  Call Extruder(12358.70300)
  MoveL 1243 to (-24.11, 11.61, 60) mm, rotated rx -180 ry 0 rz 180 deg; joints [-156.928, -57.132, -93.982, 25.942, 63.614, -12.2]
  Call Extruder(12368.06781)
  MoveL 1244 to (-26.09, 5.96, 60) mm, rotated rx -180 ry 0 rz 180 deg; joints [-157.665, -56.949, -94.65, 25.035, 63.9, -11.611]
  Call Extruder(12377.43291)
  MoveL 1245 to (-26.77, 0, 60) mm, rotated rx -180 ry 0 rz 180 deg; joints [-158.546, -56.823, -95.122, 24.004, 64.04, -11.03]
  Call Extruder(12382.22164)
  MoveL 1246 to (-26.42, -3.05, 60) mm, rotated rx -180 ry 0 rz 180 deg; joints [-159.044, -56.788, -95.251, 23.441, 64.033, -10.75]
  Set speed (130.0 mm/s)
  MoveL 1247 to (-41.86, -6.3, 60) mm, rotated rx 180 ry 0 rz 180 deg; joints [-158.606, -56.142, -97.794, 23.564, 65.852, -10.116]
  Call Extruder(12387.21949)
  Set speed (60.0 mm/s)
  MoveL 1248 to (-41.5, -9.47, 60) mm, rotated rx 180 ry 0 rz -180 deg; joints [-159.151, -56.11, -97.925, 22.957, 65.848, -9.832]
  Call Extruder(12402.11514)
  MoveL 1249 to (-38.36, -18.47, 60) mm, rotated rx -180 ry 0 rz 180 deg; joints [-160.835, -56.105, -97.945, 21.132, 65.585, -9.077]
  Call Extruder(12417.01100)
  MoveL 1250 to (-33.28, -26.54, 60) mm, rotated rx 180 ry 0 rz 180 deg; joints [-162.466, -56.194, -97.578, 19.403, 65.076, -8.443]
  Call Extruder(12431.90681)
  MoveL 1251 to (-26.54, -33.28, 60) mm, rotated rx -180 ry 0 rz -180 deg; joints [-163.93, -56.376, -96.846, 17.884, 64.347, -7.952]
  Call Extruder(12446.80266)
  MoveL 1252 to (-18.47, -38.36, 60) mm, rotated rx 180 ry 0 rz 180 deg; joints [-165.137, -56.645, -95.795, 16.666, 63.436, -7.625]
  Call Extruder(12461.69831)
  MoveL 1253 to (-9.47, -41.5, 60) mm, rotated rx 180 ry 0 rz 180 deg; joints [-166.024, -56.995, -94.483, 15.815, 62.396, -7.477]
  Call Extruder(12476.59419)
  MoveL 1254 to (0, -42.57, 60) mm, rotated rx 180 ry 0 rz 180 deg; joints [-166.562, -57.411, -92.984, 15.366, 61.283, -7.522]
  Call Extruder(12481.08976)
  MoveL 1255 to (2.86, -42.25, 60) mm, rotated rx 180 ry 0 rz 180 deg; joints [-166.618, -57.549, -92.502, 15.353, 60.943, -7.595]
  Call Extruder(12491.49006)
  MoveL 1256 to (9.47, -41.51, 60) mm, rotated rx 180 ry 0 rz 180 deg; joints [-166.745, -57.877, -91.377, 15.328, 60.158, -7.767]
  Call Extruder(12506.38572)
  MoveL 1257 to (18.47, -38.36, 60) mm, rotated rx -180 ry 0 rz 180 deg; joints [-166.591, -58.369, -89.743, 15.683, 59.079, -8.21]
  Call Extruder(12521.28157)
  MoveL 1258 to (26.54, -33.28, 60) mm, rotated rx 180 ry 0 rz 180 deg; joints [-166.133, -58.862, -88.162, 16.398, 58.102, -8.839]
  Call Extruder(12536.17739)
  MoveL 1259 to (33.29, -26.54, 60) mm, rotated rx -180 ry 0 rz 180 deg; joints [-165.409, -59.329, -86.71, 17.424, 57.275, -9.629]
  Call Extruder(12551.07324)
  MoveL 1260 to (38.36, -18.47, 60) mm, rotated rx -180 ry 0 rz -180 deg; joints [-164.468, -59.742, -85.455, 18.7, 56.639, -10.544]
  Call Extruder(12565.96889)
  MoveL 1261 to (41.5, -9.47, 60) mm, rotated rx 180 ry 0 rz 180 deg; joints [-163.355, -60.078, -84.454, 20.158, 56.225, -11.534]
  Call Extruder(12580.86476)
  MoveL 1262 to (42.57, 0, 60) mm, rotated rx 180 ry 0 rz 180 deg; joints [-162.12, -60.316, -83.753, 21.723, 56.051, -12.544]
  Call Extruder(12595.76064)
  MoveL 1263 to (41.51, 9.47, 60) mm, rotated rx 180 ry 0 rz 180 deg; joints [-160.81, -60.442, -83.386, 23.323, 56.123, -13.513]
  Call Extruder(12610.65630)
  MoveL 1264 to (38.36, 18.47, 60) mm, rotated rx -180 ry 0 rz -180 deg; joints [-159.475, -60.448, -83.368, 24.884, 56.434, -14.384]
  Call Extruder(12625.55214)
  MoveL 1265 to (33.29, 26.54, 60) mm, rotated rx 180 ry 0 rz 180 deg; joints [-158.16, -60.334, -83.702, 26.343, 56.966, -15.106]
  Call Extruder(12640.44797)
  MoveL 1266 to (26.54, 33.28, 60) mm, rotated rx 180 ry 0 rz -180 deg; joints [-156.916, -60.106, -84.37, 27.64, 57.689, -15.638]
  Call Extruder(12655.34381)
  MoveL 1267 to (18.47, 38.36, 60) mm, rotated rx 180 ry 0 rz -180 deg; joints [-155.789, -59.779, -85.343, 28.727, 58.565, -15.953]
  Call Extruder(12670.23948)
  MoveL 1268 to (9.47, 41.51, 60) mm, rotated rx 180 ry 0 rz 180 deg; joints [-154.828, -59.372, -86.576, 29.563, 59.552, -16.037]
  Call Extruder(12685.13535)
  MoveL 1269 to (0, 42.57, 60) mm, rotated rx 180 ry 0 rz 180 deg; joints [-154.081, -58.91, -88.012, 30.113, 60.601, -15.892]
  Call Extruder(12700.03122)
  MoveL 1270 to (-9.47, 41.51, 60) mm, rotated rx 180 ry 0 rz -180 deg; joints [-153.594, -58.418, -89.583, 30.349, 61.666, -15.53]
  Call Extruder(12714.92687)
  MoveL 1271 to (-18.47, 38.36, 60) mm, rotated rx 180 ry 0 rz 180 deg; joints [-153.408, -57.925, -91.215, 30.248, 62.698, -14.975]
  Call Extruder(12729.82273)
  MoveL 1272 to (-26.54, 33.29, 60) mm, rotated rx 180 ry 0 rz 180 deg; joints [-153.557, -57.456, -92.828, 29.797, 63.651, -14.261]
  Call Extruder(12744.71854)
  MoveL 1273 to (-33.28, 26.54, 60) mm, rotated rx 180 ry 0 rz -180 deg; joints [-154.059, -57.033, -94.341, 28.995, 64.481, -13.428]
  Call Extruder(12759.61439)
  MoveL 1274 to (-38.36, 18.47, 60) mm, rotated rx 180 ry 0 rz -180 deg; joints [-154.913, -56.677, -95.675, 27.857, 65.148, -12.523]
  Call Extruder(12774.51005)
  MoveL 1275 to (-41.51, 9.47, 60) mm, rotated rx 180 ry 0 rz -180 deg; joints [-156.091, -56.399, -96.755, 26.422, 65.617, -11.593]
  Call Extruder(12789.40592)
  MoveL 1276 to (-42.57, 0, 60) mm, rotated rx 180 ry 0 rz -180 deg; joints [-157.533, -56.208, -97.521, 24.758, 65.857, -10.682]
  Call Extruder(12796.96020)
  MoveL 1277 to (-42.03, -4.8, 60) mm, rotated rx 180 ry 0 rz 180 deg; joints [-158.35, -56.157, -97.731, 23.848, 65.853, -10.25]
  Set speed (130.0 mm/s)
  MoveL 1278 to (-54.1, -7.67, 60) mm, rotated rx 180 ry 0 rz 180 deg; joints [-158.024, -55.698, -99.697, 23.934, 67.287, -9.724]
  Call Extruder(12801.03283)
  Set speed (30.0 mm/s)
  MoveL 1279 to (-53.59, -12.23, 60) mm, rotated rx -180 ry 0 rz 180 deg; joints [-158.835, -55.656, -99.887, 23.042, 67.288, -9.326]
  Call Extruder(12811.96296)
  MoveL 1280 to (-49.53, -23.85, 60) mm, rotated rx 180 ry 0 rz -180 deg; joints [-161.095, -55.65, -99.912, 20.615, 66.959, -8.375]
  Call Extruder(12822.89325)
  MoveL 1281 to (-42.98, -34.27, 60) mm, rotated rx -180 ry 0 rz 180 deg; joints [-163.275, -55.758, -99.429, 18.317, 66.303, -7.579]
  Call Extruder(12833.82337)
  MoveL 1282 to (-34.27, -42.98, 60) mm, rotated rx 180 ry 0 rz -180 deg; joints [-165.21, -55.98, -98.468, 16.312, 65.352, -6.958]
  Call Extruder(12844.75365)
  MoveL 1283 to (-23.85, -49.53, 60) mm, rotated rx 180 ry 0 rz 180 deg; joints [-166.774, -56.315, -97.09, 14.727, 64.164, -6.535]
  Call Extruder(12855.68378)
  MoveL 1284 to (-12.23, -53.59, 60) mm, rotated rx 180 ry 0 rz 180 deg; joints [-167.889, -56.754, -95.38, 13.644, 62.807, -6.33]
  Call Extruder(12866.61401)
  MoveL 1285 to (0, -54.97, 60) mm, rotated rx 180 ry 0 rz 180 deg; joints [-168.526, -57.284, -93.434, 13.1, 61.358, -6.365]
  Call Extruder(12870.40133)
  MoveL 1286 to (4.24, -54.49, 60) mm, rotated rx -180 ry 0 rz 180 deg; joints [-168.587, -57.487, -92.718, 13.096, 60.852, -6.464]
  Call Extruder(12877.54423)
  MoveL 1287 to (12.23, -53.59, 60) mm, rotated rx 180 ry 0 rz 180 deg; joints [-168.697, -57.883, -91.355, 13.094, 59.898, -6.654]
  Call Extruder(12888.47437)
  MoveL 1288 to (23.85, -49.53, 60) mm, rotated rx 180 ry 0 rz 180 deg; joints [-168.436, -58.521, -89.25, 13.597, 58.501, -7.203]
  Call Extruder(12899.40465)
  MoveL 1289 to (34.27, -42.98, 60) mm, rotated rx 180 ry 0 rz 180 deg; joints [-167.797, -59.164, -87.217, 14.558, 57.238, -8]
  Call Extruder(12910.33477)
  MoveL 1290 to (42.98, -34.27, 60) mm, rotated rx -180 ry 0 rz 180 deg; joints [-166.837, -59.776, -85.354, 15.91, 56.172, -9.017]
  Call Extruder(12921.26505)
  MoveL 1291 to (49.53, -23.85, 60) mm, rotated rx 180 ry 0 rz 180 deg; joints [-165.618, -60.319, -83.744, 17.573, 55.354, -10.206]
  Call Extruder(12932.19519)
  MoveL 1292 to (53.59, -12.23, 60) mm, rotated rx 180 ry 0 rz -180 deg; joints [-164.2, -60.762, -82.461, 19.457, 54.825, -11.504]
  Call Extruder(12943.12541)
  MoveL 1293 to (54.97, 0, 60) mm, rotated rx -180 ry 0 rz 180 deg; joints [-162.641, -61.077, -81.564, 21.469, 54.608, -12.832]
  Call Extruder(12954.05563)
  MoveL 1294 to (53.59, 12.23, 60) mm, rotated rx 180 ry 0 rz -180 deg; joints [-160.996, -61.244, -81.093, 23.512, 54.71, -14.109]
  Call Extruder(12964.98577)
  MoveL 1295 to (49.52, 23.85, 60) mm, rotated rx 180 ry 0 rz -180 deg; joints [-159.322, -61.252, -81.071, 25.495, 55.121, -15.253]
  Call Extruder(12975.91605)
  MoveL 1296 to (42.98, 34.27, 60) mm, rotated rx -180 ry 0 rz 180 deg; joints [-157.673, -61.1, -81.498, 27.338, 55.815, -16.197]
  Call Extruder(12986.84617)
  MoveL 1297 to (34.27, 42.98, 60) mm, rotated rx 180 ry 0 rz 180 deg; joints [-156.102, -60.8, -82.354, 28.973, 56.752, -16.887]
  Call Extruder(12997.77645)
  MoveL 1298 to (23.85, 49.52, 60) mm, rotated rx 180 ry 0 rz 180 deg; joints [-154.667, -60.368, -83.601, 30.344, 57.883, -17.287]
  Call Extruder(13008.70659)
  MoveL 1299 to (12.23, 53.59, 60) mm, rotated rx -180 ry 0 rz 180 deg; joints [-153.426, -59.833, -85.181, 31.405, 59.15, -17.384]
  Call Extruder(13019.63681)
  MoveL 1300 to (0, 54.97, 60) mm, rotated rx 180 ry 0 rz 180 deg; joints [-152.438, -59.227, -87.023, 32.118, 60.494, -17.18]
  Call Extruder(13030.56704)
  MoveL 1301 to (-12.23, 53.59, 60) mm, rotated rx 180 ry 0 rz 180 deg; joints [-151.764, -58.585, -89.043, 32.449, 61.856, -16.695]
  Call Extruder(13041.49717)
  MoveL 1302 to (-23.85, 49.52, 60) mm, rotated rx 180 ry 0 rz 180 deg; joints [-151.463, -57.945, -91.146, 32.366, 63.175, -15.961]
  Call Extruder(13052.42745)
  MoveL 1303 to (-34.27, 42.98, 60) mm, rotated rx -180 ry 0 rz 180 deg; joints [-151.589, -57.341, -93.232, 31.843, 64.397, -15.023]
  Call Extruder(13063.35757)
  MoveL 1304 to (-42.98, 34.27, 60) mm, rotated rx 180 ry 0 rz -180 deg; joints [-152.179, -56.803, -95.196, 30.865, 65.467, -13.937]
  Call Extruder(13074.28785)
  MoveL 1305 to (-49.52, 23.85, 60) mm, rotated rx 180 ry 0 rz 180 deg; joints [-153.248, -56.354, -96.934, 29.437, 66.335, -12.763]
  Call Extruder(13085.21799)
  MoveL 1306 to (-53.59, 12.23, 60) mm, rotated rx -180 ry 0 rz 180 deg; joints [-154.769, -56.009, -98.348, 27.596, 66.954, -11.565]
  Call Extruder(13096.14821)
  MoveL 1307 to (-54.97, 0, 60) mm, rotated rx 180 ry 0 rz -180 deg; joints [-156.673, -55.775, -99.354, 25.423, 67.282, -10.402]
  Call Extruder(13101.67383)
  MoveL 1308 to (-54.27, -6.18, 60) mm, rotated rx 180 ry 0 rz -180 deg; joints [-157.76, -55.712, -99.633, 24.224, 67.287, -9.855]
  Set speed (130.0 mm/s)
  MoveL 1309 to (-49.9, -9.51, 60) mm, rotated rx 180 ry 0 rz 180 deg; joints [-158.616, -55.814, -99.183, 23.367, 66.823, -9.65]
  MoveL 1310 to (2.97, -12.99, 60) mm, rotated rx 180 ry 0 rz -180 deg; joints [-162.152, -57.947, -91.141, 20.571, 60.725, -10.399]
  Call Extruder(13106.33740)
  Set speed (80.0 mm/s)
  MoveL 1311 to (5.78, -12.01, 60) mm, rotated rx 180 ry 0 rz -180 deg; joints [-162.141, -58.1, -90.629, 20.655, 60.391, -10.551]
  Call Extruder(13111.00102)
  MoveL 1312 to (8.31, -10.42, 60) mm, rotated rx 180 ry 0 rz -180 deg; joints [-162.027, -58.251, -90.129, 20.855, 60.086, -10.757]
  Call Extruder(13115.66521)
  MoveL 1313 to (10.42, -8.31, 60) mm, rotated rx -180 ry 0 rz 180 deg; joints [-161.819, -58.392, -89.668, 21.157, 59.827, -11.007]
  Call Extruder(13120.32884)
  MoveL 1314 to (12.01, -5.78, 60) mm, rotated rx 180 ry 0 rz 180 deg; joints [-161.529, -58.516, -89.267, 21.546, 59.625, -11.291]
  Call Extruder(13124.99241)
  MoveL 1315 to (12.99, -2.97, 60) mm, rotated rx 180 ry 0 rz -180 deg; joints [-161.171, -58.615, -88.947, 22, 59.491, -11.592]
  Call Extruder(13129.65636)
  MoveL 1316 to (13.33, 0, 60) mm, rotated rx -180 ry 0 rz 180 deg; joints [-160.763, -58.686, -88.723, 22.499, 59.431, -11.895]
  Call Extruder(13134.32032)
  MoveL 1317 to (12.99, 2.97, 60) mm, rotated rx 180 ry 0 rz 180 deg; joints [-160.324, -58.723, -88.605, 23.016, 59.448, -12.185]
  Call Extruder(13138.98389)
  MoveL 1318 to (12.01, 5.78, 60) mm, rotated rx -180 ry 0 rz -180 deg; joints [-159.874, -58.724, -88.599, 23.527, 59.541, -12.446]
  Call Extruder(13143.64751)
  MoveL 1319 to (10.42, 8.31, 60) mm, rotated rx -180 ry 0 rz 180 deg; joints [-159.432, -58.691, -88.706, 24.009, 59.704, -12.664]
  Call Extruder(13148.31170)
  MoveL 1320 to (8.31, 10.42, 60) mm, rotated rx -180 ry 0 rz 180 deg; joints [-159.021, -58.624, -88.92, 24.438, 59.929, -12.828]
  Call Extruder(13152.97533)
  MoveL 1321 to (5.78, 12.01, 60) mm, rotated rx 180 ry 0 rz 180 deg; joints [-158.657, -58.527, -89.232, 24.796, 60.205, -12.929]
  Call Extruder(13157.63890)
  MoveL 1322 to (2.97, 12.99, 60) mm, rotated rx -180 ry 0 rz 180 deg; joints [-158.359, -58.405, -89.625, 25.065, 60.518, -12.962]
  Call Extruder(13162.30285)
  MoveL 1323 to (0, 13.33, 60) mm, rotated rx -180 ry 0 rz 180 deg; joints [-158.143, -58.266, -90.082, 25.231, 60.853, -12.926]
  Call Extruder(13166.96681)
  MoveL 1324 to (-2.97, 12.99, 60) mm, rotated rx 180 ry 0 rz 180 deg; joints [-158.019, -58.115, -90.578, 25.287, 61.194, -12.824]
  Call Extruder(13171.63038)
  MoveL 1325 to (-5.78, 12.01, 60) mm, rotated rx 180 ry 0 rz -180 deg; joints [-157.997, -57.962, -91.091, 25.228, 61.524, -12.661]
  Call Extruder(13176.29401)
  MoveL 1326 to (-8.31, 10.42, 60) mm, rotated rx 180 ry 0 rz 180 deg; joints [-158.08, -57.813, -91.593, 25.055, 61.826, -12.447]
  Call Extruder(13180.95820)
  MoveL 1327 to (-10.42, 8.31, 60) mm, rotated rx 180 ry 0 rz 180 deg; joints [-158.266, -57.677, -92.061, 24.774, 62.086, -12.192]
  Call Extruder(13185.62182)
  MoveL 1328 to (-12.01, 5.78, 60) mm, rotated rx 180 ry 0 rz -180 deg; joints [-158.549, -57.558, -92.469, 24.399, 62.291, -11.91]
  Call Extruder(13190.28539)
  MoveL 1329 to (-12.99, 2.97, 60) mm, rotated rx 180 ry 0 rz -180 deg; joints [-158.913, -57.464, -92.797, 23.946, 62.431, -11.615]
  Call Extruder(13194.94935)
  MoveL 1330 to (-13.33, 0, 60) mm, rotated rx 180 ry 0 rz -180 deg; joints [-159.341, -57.399, -93.028, 23.438, 62.497, -11.321]
  Call Extruder(13199.61330)
  MoveL 1331 to (-12.99, -2.97, 60) mm, rotated rx 180 ry 0 rz 180 deg; joints [-159.811, -57.364, -93.15, 22.901, 62.486, -11.042]
  Call Extruder(13204.27687)
  MoveL 1332 to (-12.01, -5.78, 60) mm, rotated rx 180 ry 0 rz -180 deg; joints [-160.294, -57.363, -93.156, 22.364, 62.398, -10.793]
  Call Extruder(13208.94050)
  MoveL 1333 to (-10.42, -8.31, 60) mm, rotated rx 180 ry 0 rz -180 deg; joints [-160.766, -57.394, -93.045, 21.856, 62.238, -10.583]
  Call Extruder(13213.60468)
  MoveL 1334 to (-8.31, -10.42, 60) mm, rotated rx 180 ry 0 rz -180 deg; joints [-161.2, -57.457, -92.825, 21.405, 62.012, -10.423]
  Call Extruder(13218.26832)
  MoveL 1335 to (-5.78, -12.01, 60) mm, rotated rx 180 ry 0 rz 180 deg; joints [-161.572, -57.548, -92.506, 21.034, 61.732, -10.322]
  Call Extruder(13222.93188)
  MoveL 1336 to (-2.97, -13, 60) mm, rotated rx 180 ry 0 rz 180 deg; joints [-161.863, -57.664, -92.104, 20.764, 61.414, -10.282]
  Call Extruder(13227.59582)
  MoveL 1337 to (0, -13.33, 60) mm, rotated rx -180 ry 0 rz -180 deg; joints [-162.059, -57.799, -91.642, 20.607, 61.072, -10.308]
  Call Extruder(13232.25979)
  MoveL 1338 to (2.97, -12.99, 60) mm, rotated rx 180 ry 0 rz -180 deg; joints [-162.152, -57.947, -91.141, 20.571, 60.725, -10.399]
  Set speed (130.0 mm/s)
  MoveL 1339 to (2.97, -12.99, 65) mm, rotated rx -180 ry 0 rz -180 deg; joints [-162.152, -57.18, -91.526, 20.647, 60.368, -10.553]
  MoveL 1340 to (-26.25, -4.54, 65) mm, rotated rx -180 ry 0 rz 180 deg; joints [-159.288, -55.977, -95.706, 23.243, 63.66, -10.789]
  Call Extruder(13234.49242)
  Set speed (60.0 mm/s)
  MoveL 1341 to (-26.09, -5.96, 65) mm, rotated rx 180 ry 0 rz 180 deg; joints [-159.522, -55.961, -95.763, 22.979, 63.655, -10.657]
  Call Extruder(13243.85722)
  MoveL 1342 to (-24.12, -11.61, 65) mm, rotated rx 180 ry 0 rz 180 deg; joints [-160.532, -55.958, -95.775, 21.869, 63.481, -10.16]
  Call Extruder(13253.22213)
  MoveL 1343 to (-20.93, -16.69, 65) mm, rotated rx 180 ry 0 rz -180 deg; joints [-161.513, -56.02, -95.549, 20.817, 63.158, -9.741]
  Call Extruder(13262.58734)
  MoveL 1344 to (-16.69, -20.93, 65) mm, rotated rx 180 ry 0 rz 180 deg; joints [-162.406, -56.144, -95.098, 19.886, 62.702, -9.419]
  Call Extruder(13271.95226)
  MoveL 1345 to (-11.61, -24.12, 65) mm, rotated rx 180 ry 0 rz 180 deg; joints [-163.159, -56.325, -94.447, 19.129, 62.138, -9.207]
  Call Extruder(13281.31705)
  MoveL 1346 to (-5.96, -26.09, 65) mm, rotated rx 180 ry 0 rz -180 deg; joints [-163.733, -56.558, -93.631, 18.587, 61.495, -9.118]
  Call Extruder(13290.68216)
  MoveL 1347 to (0, -26.77, 65) mm, rotated rx 180 ry 0 rz -180 deg; joints [-164.103, -56.831, -92.694, 18.286, 60.806, -9.156]
  Call Extruder(13293.06822)
  MoveL 1348 to (1.52, -26.59, 65) mm, rotated rx 180 ry 0 rz -180 deg; joints [-164.143, -56.907, -92.438, 18.273, 60.629, -9.199]
  Call Extruder(13300.04726)
  MoveL 1349 to (5.96, -26.09, 65) mm, rotated rx 180 ry 0 rz 180 deg; joints [-164.258, -57.133, -91.685, 18.236, 60.109, -9.325]
  Call Extruder(13309.41206)
  MoveL 1350 to (11.61, -24.11, 65) mm, rotated rx 180 ry 0 rz 180 deg; joints [-164.201, -57.447, -90.654, 18.433, 59.439, -9.618]
  Call Extruder(13318.77697)
  MoveL 1351 to (16.69, -20.93, 65) mm, rotated rx -180 ry 0 rz 180 deg; joints [-163.944, -57.76, -89.654, 18.859, 58.831, -10.026]
  Call Extruder(13328.14218)
  MoveL 1352 to (20.93, -16.69, 65) mm, rotated rx 180 ry 0 rz 180 deg; joints [-163.508, -58.053, -88.733, 19.488, 58.316, -10.529]
  Call Extruder(13337.50710)
  MoveL 1353 to (24.12, -11.61, 65) mm, rotated rx 180 ry 0 rz 180 deg; joints [-162.92, -58.311, -87.934, 20.283, 57.918, -11.105]
  Call Extruder(13346.87189)
  MoveL 1354 to (26.09, -5.96, 65) mm, rotated rx -180 ry 0 rz -180 deg; joints [-162.209, -58.52, -87.297, 21.201, 57.659, -11.723]
  Call Extruder(13356.23700)
  MoveL 1355 to (26.77, 0, 65) mm, rotated rx -180 ry 0 rz -180 deg; joints [-161.41, -58.668, -86.851, 22.197, 57.548, -12.35]
  Call Extruder(13365.60210)
  MoveL 1356 to (26.09, 5.96, 65) mm, rotated rx 180 ry 0 rz 180 deg; joints [-160.556, -58.746, -86.617, 23.222, 57.591, -12.951]
  Call Extruder(13374.96690)
  MoveL 1357 to (24.12, 11.61, 65) mm, rotated rx 180 ry 0 rz 180 deg; joints [-159.683, -58.75, -86.606, 24.23, 57.784, -13.492]
  Call Extruder(13384.33181)
  MoveL 1358 to (20.93, 16.69, 65) mm, rotated rx 180 ry 0 rz 180 deg; joints [-158.826, -58.679, -86.818, 25.176, 58.116, -13.943]
  Call Extruder(13393.69702)
  MoveL 1359 to (16.69, 20.93, 65) mm, rotated rx -180 ry 0 rz 180 deg; joints [-158.019, -58.538, -87.244, 26.018, 58.569, -14.281]
  Call Extruder(13403.06194)
  MoveL 1360 to (11.61, 24.11, 65) mm, rotated rx 180 ry 0 rz -180 deg; joints [-157.299, -58.335, -87.863, 26.722, 59.121, -14.487]
  Call Extruder(13412.42674)
  MoveL 1361 to (5.96, 26.09, 65) mm, rotated rx -180 ry 0 rz 180 deg; joints [-156.697, -58.081, -88.647, 27.257, 59.744, -14.552]
  Call Extruder(13421.79184)
  MoveL 1362 to (0, 26.77, 65) mm, rotated rx -180 ry 0 rz 180 deg; joints [-156.245, -57.79, -89.558, 27.597, 60.408, -14.474]
  Call Extruder(13431.15695)
  MoveL 1363 to (-5.96, 26.09, 65) mm, rotated rx 180 ry 0 rz 180 deg; joints [-155.969, -57.479, -90.553, 27.726, 61.082, -14.26]
  Call Extruder(13440.52174)
  MoveL 1364 to (-11.61, 24.12, 65) mm, rotated rx 180 ry 0 rz 180 deg; joints [-155.891, -57.163, -91.582, 27.631, 61.733, -13.923]
  Call Extruder(13449.88666)
  MoveL 1365 to (-16.69, 20.93, 65) mm, rotated rx 180 ry 0 rz -180 deg; joints [-156.025, -56.86, -92.596, 27.31, 62.332, -13.483]
  Call Extruder(13459.25187)
  MoveL 1366 to (-20.93, 16.69, 65) mm, rotated rx 180 ry 0 rz -180 deg; joints [-156.374, -56.583, -93.543, 26.77, 62.849, -12.964]
  Call Extruder(13468.61678)
  MoveL 1367 to (-24.11, 11.61, 65) mm, rotated rx -180 ry 0 rz 180 deg; joints [-156.928, -56.346, -94.373, 26.029, 63.258, -12.394]
  Call Extruder(13477.98158)
  MoveL 1368 to (-26.09, 5.96, 65) mm, rotated rx -180 ry 0 rz -180 deg; joints [-157.665, -56.159, -95.042, 25.119, 63.538, -11.8]
  Call Extruder(13487.34669)
  MoveL 1369 to (-26.77, 0, 65) mm, rotated rx -180 ry 0 rz 180 deg; joints [-158.546, -56.029, -95.514, 24.084, 63.674, -11.212]
  Call Extruder(13492.13541)
  MoveL 1370 to (-26.42, -3.05, 65) mm, rotated rx 180 ry 0 rz -180 deg; joints [-159.044, -55.994, -95.644, 23.52, 63.665, -10.928]
  Set speed (130.0 mm/s)
  MoveL 1371 to (-41.86, -6.29, 65) mm, rotated rx 180 ry 0 rz 180 deg; joints [-158.606, -55.328, -98.193, 23.639, 65.471, -10.299]
  Call Extruder(13497.13327)
  Set speed (60.0 mm/s)
  MoveL 1372 to (-41.51, -9.47, 65) mm, rotated rx -180 ry 0 rz 180 deg; joints [-159.151, -55.295, -98.325, 23.031, 65.466, -10.011]
  Call Extruder(13512.02892)
  MoveL 1373 to (-38.36, -18.47, 65) mm, rotated rx 180 ry 0 rz -180 deg; joints [-160.835, -55.29, -98.344, 21.201, 65.198, -9.242]
  Call Extruder(13526.92477)
  MoveL 1374 to (-33.28, -26.54, 65) mm, rotated rx 180 ry 0 rz 180 deg; joints [-162.466, -55.382, -97.976, 19.468, 64.686, -8.595]
  Call Extruder(13541.82058)
  MoveL 1375 to (-26.54, -33.28, 65) mm, rotated rx 180 ry 0 rz -180 deg; joints [-163.93, -55.569, -97.243, 17.945, 63.956, -8.093]
  Call Extruder(13556.71644)
  MoveL 1376 to (-18.47, -38.36, 65) mm, rotated rx 180 ry 0 rz 180 deg; joints [-165.137, -55.847, -96.189, 16.724, 63.048, -7.755]
  Call Extruder(13571.61209)
  MoveL 1377 to (-9.47, -41.51, 65) mm, rotated rx 180 ry 0 rz -180 deg; joints [-166.024, -56.206, -94.874, 15.872, 62.013, -7.6]
  Call Extruder(13586.50797)
  MoveL 1378 to (0, -42.57, 65) mm, rotated rx 180 ry 0 rz 180 deg; joints [-166.562, -56.633, -93.372, 15.423, 60.906, -7.64]
  Call Extruder(13591.65957)
  MoveL 1379 to (3.28, -42.2, 65) mm, rotated rx 180 ry 0 rz 180 deg; joints [-166.626, -56.795, -92.818, 15.409, 60.52, -7.724]
  Call Extruder(13601.40384)
  MoveL 1380 to (9.47, -41.51, 65) mm, rotated rx 180 ry 0 rz 180 deg; joints [-166.745, -57.109, -91.762, 15.386, 59.789, -7.884]
  Call Extruder(13616.29950)
  MoveL 1381 to (18.47, -38.36, 65) mm, rotated rx -180 ry 0 rz 180 deg; joints [-166.591, -57.612, -90.126, 15.744, 58.718, -8.328]
  Call Extruder(13631.19534)
  MoveL 1382 to (26.54, -33.28, 65) mm, rotated rx 180 ry 0 rz 180 deg; joints [-166.133, -58.114, -88.543, 16.463, 57.749, -8.961]
  Call Extruder(13646.09116)
  MoveL 1383 to (33.28, -26.54, 65) mm, rotated rx 180 ry 0 rz 180 deg; joints [-165.409, -58.589, -87.089, 17.494, 56.93, -9.758]
  Call Extruder(13660.98702)
  MoveL 1384 to (38.36, -18.47, 65) mm, rotated rx 180 ry 0 rz 180 deg; joints [-164.468, -59.009, -85.832, 18.776, 56.302, -10.681]
  Call Extruder(13675.88267)
  MoveL 1385 to (41.5, -9.47, 65) mm, rotated rx -180 ry 0 rz 180 deg; joints [-163.355, -59.35, -84.83, 20.239, 55.895, -11.681]
  Call Extruder(13690.77854)
  MoveL 1386 to (42.57, 0, 65) mm, rotated rx 180 ry 0 rz -180 deg; joints [-162.12, -59.592, -84.129, 21.811, 55.727, -12.7]
  Call Extruder(13705.67441)
  MoveL 1387 to (41.5, 9.47, 65) mm, rotated rx -180 ry 0 rz 180 deg; joints [-160.81, -59.72, -83.762, 23.415, 55.805, -13.679]
  Call Extruder(13720.57008)
  MoveL 1388 to (38.36, 18.47, 65) mm, rotated rx -180 ry 0 rz 180 deg; joints [-159.475, -59.726, -83.744, 24.982, 56.12, -14.56]
  Call Extruder(13735.46592)
  MoveL 1389 to (33.28, 26.54, 65) mm, rotated rx -180 ry 0 rz 180 deg; joints [-158.16, -59.61, -84.078, 26.444, 56.655, -15.29]
  Call Extruder(13750.36174)
  MoveL 1390 to (26.54, 33.28, 65) mm, rotated rx -180 ry 0 rz 180 deg; joints [-156.916, -59.379, -84.747, 27.744, 57.379, -15.831]
  Call Extruder(13765.25759)
  MoveL 1391 to (18.47, 38.36, 65) mm, rotated rx 180 ry 0 rz -180 deg; joints [-155.789, -59.047, -85.721, 28.832, 58.254, -16.153]
  Call Extruder(13780.15325)
  MoveL 1392 to (9.47, 41.51, 65) mm, rotated rx 180 ry 0 rz -180 deg; joints [-154.828, -58.634, -86.955, 29.668, 59.238, -16.244]
  Call Extruder(13795.04912)
  MoveL 1393 to (0, 42.57, 65) mm, rotated rx 180 ry 0 rz -180 deg; joints [-154.081, -58.163, -88.392, 30.218, 60.284, -16.104]
  Call Extruder(13809.94500)
  MoveL 1394 to (-9.47, 41.51, 65) mm, rotated rx -180 ry 0 rz -180 deg; joints [-153.594, -57.662, -89.965, 30.451, 61.343, -15.745]
  Call Extruder(13824.84065)
  MoveL 1395 to (-18.47, 38.36, 65) mm, rotated rx 180 ry 0 rz 180 deg; joints [-153.408, -57.158, -91.6, 30.348, 62.368, -15.192]
  Call Extruder(13839.73650)
  MoveL 1396 to (-26.54, 33.29, 65) mm, rotated rx -180 ry 0 rz 180 deg; joints [-153.557, -56.678, -93.216, 29.894, 63.313, -14.477]
  Call Extruder(13854.63232)
  MoveL 1397 to (-33.28, 26.54, 65) mm, rotated rx -180 ry 0 rz 180 deg; joints [-154.059, -56.245, -94.732, 29.088, 64.134, -13.642]
  Call Extruder(13869.52817)
  MoveL 1398 to (-38.36, 18.47, 65) mm, rotated rx 180 ry 0 rz -180 deg; joints [-154.913, -55.879, -96.069, 27.945, 64.791, -12.732]
  Call Extruder(13884.42383)
  MoveL 1399 to (-41.5, 9.47, 65) mm, rotated rx 180 ry 0 rz 180 deg; joints [-156.091, -55.593, -97.152, 26.506, 65.25, -11.793]
  Call Extruder(13899.31970)
  MoveL 1400 to (-42.57, 0, 65) mm, rotated rx -180 ry 0 rz -180 deg; joints [-157.533, -55.396, -97.919, 24.836, 65.481, -10.873]
  Call Extruder(13906.87397)
  MoveL 1401 to (-42.03, -4.8, 65) mm, rotated rx -180 ry 0 rz 180 deg; joints [-158.35, -55.343, -98.13, 23.924, 65.474, -10.434]
  Set speed (130.0 mm/s)
  MoveL 1402 to (-54.1, -7.67, 65) mm, rotated rx -180 ry 0 rz 180 deg; joints [-158.024, -54.868, -100.101, 24.007, 66.899, -9.912]
  Call Extruder(13910.94661)
  Set speed (30.0 mm/s)
  MoveL 1403 to (-53.59, -12.23, 65) mm, rotated rx -180 ry 0 rz 180 deg; joints [-158.835, -54.824, -100.292, 23.112, 66.896, -9.507]
  Call Extruder(13921.87674)
  MoveL 1404 to (-49.52, -23.85, 65) mm, rotated rx 180 ry 0 rz 180 deg; joints [-161.095, -54.819, -100.317, 20.68, 66.56, -8.539]
  Call Extruder(13932.80702)
  MoveL 1405 to (-42.98, -34.27, 65) mm, rotated rx 180 ry 0 rz 180 deg; joints [-163.275, -54.931, -99.832, 18.376, 65.9, -7.725]
  Call Extruder(13943.73714)
  MoveL 1406 to (-34.27, -42.98, 65) mm, rotated rx 180 ry 0 rz -180 deg; joints [-165.21, -55.161, -98.868, 16.366, 64.95, -7.088]
  Call Extruder(13954.66743)
  MoveL 1407 to (-23.85, -49.53, 65) mm, rotated rx 180 ry 0 rz 180 deg; joints [-166.774, -55.506, -97.488, 14.778, 63.766, -6.651]
  Call Extruder(13965.59756)
  MoveL 1408 to (-12.23, -53.59, 65) mm, rotated rx -180 ry 0 rz 180 deg; joints [-167.889, -55.959, -95.773, 13.693, 62.415, -6.437]
  Call Extruder(13976.52778)
  MoveL 1409 to (0, -54.97, 65) mm, rotated rx -180 ry 0 rz 180 deg; joints [-168.526, -56.503, -93.823, 13.149, 60.976, -6.466]
  Call Extruder(13980.68794)
  MoveL 1410 to (4.65, -54.44, 65) mm, rotated rx -180 ry 0 rz 180 deg; joints [-168.593, -56.731, -93.035, 13.145, 60.424, -6.575]
  Call Extruder(13987.45800)
  MoveL 1411 to (12.23, -53.59, 65) mm, rotated rx 180 ry 0 rz 180 deg; joints [-168.697, -57.116, -91.741, 13.145, 59.525, -6.755]
  Call Extruder(13998.38814)
  MoveL 1412 to (23.85, -49.53, 65) mm, rotated rx -180 ry 0 rz 180 deg; joints [-168.436, -57.767, -89.632, 13.651, 58.139, -7.306]
  Call Extruder(14009.31842)
  MoveL 1413 to (34.27, -42.98, 65) mm, rotated rx -180 ry 0 rz 180 deg; joints [-167.797, -58.422, -87.597, 14.617, 56.887, -8.109]
  Call Extruder(14020.24854)
  MoveL 1414 to (42.98, -34.27, 65) mm, rotated rx -180 ry 0 rz 180 deg; joints [-166.837, -59.043, -85.731, 15.975, 55.831, -9.134]
  Call Extruder(14031.17883)
  MoveL 1415 to (49.52, -23.85, 65) mm, rotated rx -180 ry 0 rz 180 deg; joints [-165.618, -59.596, -84.12, 17.646, 55.023, -10.334]
  Call Extruder(14042.10896)
  MoveL 1416 to (53.59, -12.23, 65) mm, rotated rx -180 ry 0 rz -180 deg; joints [-164.2, -60.045, -82.836, 19.538, 54.502, -11.644]
  Call Extruder(14053.03918)
  MoveL 1417 to (54.97, 0, 65) mm, rotated rx 180 ry 0 rz 180 deg; joints [-162.641, -60.364, -81.939, 21.558, 54.293, -12.985]
  Call Extruder(14063.96940)
  MoveL 1418 to (53.59, 12.23, 65) mm, rotated rx 180 ry 0 rz 180 deg; joints [-160.996, -60.532, -81.468, 23.608, 54.401, -14.274]
  Call Extruder(14074.89955)
  MoveL 1419 to (49.52, 23.85, 65) mm, rotated rx 180 ry 0 rz -180 deg; joints [-159.322, -60.541, -81.445, 25.597, 54.817, -15.431]
  Call Extruder(14085.82982)
  MoveL 1420 to (42.98, 34.27, 65) mm, rotated rx -180 ry 0 rz 180 deg; joints [-157.673, -60.387, -81.872, 27.445, 55.515, -16.386]
  Call Extruder(14096.75995)
  MoveL 1421 to (34.27, 42.98, 65) mm, rotated rx 180 ry 0 rz 180 deg; joints [-156.102, -60.083, -82.729, 29.082, 56.453, -17.085]
  Call Extruder(14107.69022)
  MoveL 1422 to (23.85, 49.52, 65) mm, rotated rx -180 ry 0 rz 180 deg; joints [-154.667, -59.645, -83.977, 30.455, 57.583, -17.495]
  Call Extruder(14118.62037)
  MoveL 1423 to (12.23, 53.59, 65) mm, rotated rx -180 ry 0 rz 180 deg; joints [-153.426, -59.102, -85.558, 31.516, 58.848, -17.599]
  Call Extruder(14129.55059)
  MoveL 1424 to (0, 54.97, 65) mm, rotated rx -180 ry 0 rz -180 deg; joints [-152.438, -58.486, -87.403, 32.228, 60.187, -17.402]
  Call Extruder(14140.48081)
  MoveL 1425 to (-12.23, 53.59, 65) mm, rotated rx -180 ry 0 rz 180 deg; joints [-151.764, -57.832, -89.425, 32.556, 61.542, -16.921]
  Call Extruder(14151.41095)
  MoveL 1426 to (-23.85, 49.52, 65) mm, rotated rx 180 ry 0 rz 180 deg; joints [-151.463, -57.179, -91.531, 32.47, 62.853, -16.19]
  Call Extruder(14162.34123)
  MoveL 1427 to (-34.27, 42.98, 65) mm, rotated rx 180 ry 0 rz 180 deg; joints [-151.589, -56.561, -93.62, 31.943, 64.064, -15.253]
  Call Extruder(14173.27135)
  MoveL 1428 to (-42.98, 34.27, 65) mm, rotated rx -180 ry 0 rz -180 deg; joints [-152.179, -56.009, -95.589, 30.96, 65.122, -14.164]
  Call Extruder(14184.20163)
  MoveL 1429 to (-49.52, 23.85, 65) mm, rotated rx -180 ry 0 rz 180 deg; joints [-153.248, -55.547, -97.331, 29.526, 65.977, -12.984]
  Call Extruder(14195.13177)
  MoveL 1430 to (-53.59, 12.23, 65) mm, rotated rx 180 ry 0 rz 180 deg; joints [-154.769, -55.19, -98.749, 27.679, 66.583, -11.776]
  Call Extruder(14206.06199)
  MoveL 1431 to (-54.97, 0, 65) mm, rotated rx 180 ry 0 rz -180 deg; joints [-156.673, -54.948, -99.757, 25.5, 66.899, -10.599]
  Call Extruder(14211.58760)
  MoveL 1432 to (-54.27, -6.18, 65) mm, rotated rx 180 ry 0 rz 180 deg; joints [-157.76, -54.883, -100.037, 24.298, 66.899, -10.045]
  Set speed (130.0 mm/s)
  MoveL 1433 to (-49.9, -9.51, 65) mm, rotated rx -180 ry 0 rz 180 deg; joints [-158.616, -54.989, -99.586, 23.439, 66.436, -9.833]
  MoveL 1434 to (0.02, -13.33, 65) mm, rotated rx 180 ry 0 rz -180 deg; joints [-162.06, -57.03, -92.024, 20.682, 60.71, -10.464]
  Call Extruder(14216.21621)
  Set speed (80.0 mm/s)
  MoveL 1435 to (2.97, -12.99, 65) mm, rotated rx -180 ry 0 rz -180 deg; joints [-162.152, -57.18, -91.526, 20.647, 60.368, -10.553]
  Call Extruder(14220.87978)
  MoveL 1436 to (5.78, -12.01, 65) mm, rotated rx 180 ry 0 rz -180 deg; joints [-162.141, -57.337, -91.013, 20.732, 60.037, -10.705]
  Call Extruder(14225.54340)
  MoveL 1437 to (8.31, -10.42, 65) mm, rotated rx -180 ry 0 rz -180 deg; joints [-162.027, -57.491, -90.513, 20.932, 59.735, -10.912]
  Call Extruder(14230.20760)
  MoveL 1438 to (10.42, -8.31, 65) mm, rotated rx 180 ry 0 rz -180 deg; joints [-161.819, -57.635, -90.051, 21.236, 59.478, -11.164]
  Call Extruder(14234.87123)
  MoveL 1439 to (12.01, -5.78, 65) mm, rotated rx 180 ry 0 rz 180 deg; joints [-161.529, -57.761, -89.649, 21.627, 59.278, -11.45]
  Call Extruder(14239.53479)
  MoveL 1440 to (12.99, -2.97, 65) mm, rotated rx 180 ry 0 rz -180 deg; joints [-161.171, -57.863, -89.329, 22.083, 59.147, -11.754]
  Call Extruder(14244.19875)
  MoveL 1441 to (13.33, 0, 65) mm, rotated rx -180 ry 0 rz -180 deg; joints [-160.763, -57.934, -89.104, 22.583, 59.089, -12.06]
  Call Extruder(14248.86270)
  MoveL 1442 to (12.99, 2.97, 65) mm, rotated rx 180 ry 0 rz 180 deg; joints [-160.324, -57.972, -88.986, 23.102, 59.108, -12.353]
  Call Extruder(14253.52628)
  MoveL 1443 to (12.01, 5.78, 65) mm, rotated rx 180 ry 0 rz -180 deg; joints [-159.874, -57.974, -88.98, 23.615, 59.202, -12.618]
  Call Extruder(14258.18990)
  MoveL 1444 to (10.42, 8.31, 65) mm, rotated rx -180 ry 0 rz 180 deg; joints [-159.432, -57.94, -89.087, 24.098, 59.366, -12.839]
  Call Extruder(14262.85409)
  MoveL 1445 to (8.31, 10.42, 65) mm, rotated rx -180 ry 0 rz 180 deg; joints [-159.021, -57.871, -89.302, 24.528, 59.591, -13.006]
  Call Extruder(14267.51771)
  MoveL 1446 to (5.78, 12.01, 65) mm, rotated rx 180 ry 0 rz 180 deg; joints [-158.657, -57.772, -89.614, 24.886, 59.867, -13.109]
  Call Extruder(14272.18129)
  MoveL 1447 to (2.97, 12.99, 65) mm, rotated rx 180 ry 0 rz 180 deg; joints [-158.359, -57.649, -90.008, 25.155, 60.179, -13.145]
  Call Extruder(14276.84524)
  MoveL 1448 to (0, 13.33, 65) mm, rotated rx 180 ry 0 rz 180 deg; joints [-158.143, -57.506, -90.465, 25.322, 60.513, -13.111]
  Call Extruder(14281.50920)
  MoveL 1449 to (-2.97, 12.99, 65) mm, rotated rx 180 ry 0 rz 180 deg; joints [-158.019, -57.353, -90.962, 25.377, 60.852, -13.009]
  Call Extruder(14286.17277)
  MoveL 1450 to (-5.78, 12.01, 65) mm, rotated rx 180 ry 0 rz -180 deg; joints [-157.997, -57.196, -91.475, 25.317, 61.179, -12.847]
  Call Extruder(14290.83639)
  MoveL 1451 to (-8.31, 10.42, 65) mm, rotated rx 180 ry 0 rz 180 deg; joints [-158.08, -57.044, -91.979, 25.143, 61.479, -12.631]
  Call Extruder(14295.50058)
  MoveL 1452 to (-10.42, 8.31, 65) mm, rotated rx -180 ry 0 rz 180 deg; joints [-158.266, -56.904, -92.447, 24.861, 61.736, -12.375]
  Call Extruder(14300.16421)
  MoveL 1453 to (-12.01, 5.78, 65) mm, rotated rx 180 ry 0 rz -180 deg; joints [-158.549, -56.783, -92.856, 24.484, 61.938, -12.091]
  Call Extruder(14304.82778)
  MoveL 1454 to (-12.99, 2.97, 65) mm, rotated rx -180 ry 0 rz -180 deg; joints [-158.913, -56.687, -93.185, 24.029, 62.075, -11.793]
  Call Extruder(14309.49174)
  MoveL 1455 to (-13.33, 0, 65) mm, rotated rx 180 ry 0 rz 180 deg; joints [-159.341, -56.62, -93.416, 23.519, 62.139, -11.497]
  Call Extruder(14314.15569)
  MoveL 1456 to (-12.99, -2.97, 65) mm, rotated rx 180 ry 0 rz 180 deg; joints [-159.811, -56.585, -93.538, 22.981, 62.126, -11.215]
  Call Extruder(14318.81926)
  MoveL 1457 to (-12.01, -5.78, 65) mm, rotated rx 180 ry 0 rz -180 deg; joints [-160.294, -56.583, -93.544, 22.443, 62.037, -10.961]
  Call Extruder(14323.48288)
  MoveL 1458 to (-10.42, -8.31, 65) mm, rotated rx 180 ry 0 rz 180 deg; joints [-160.766, -56.615, -93.434, 21.933, 61.875, -10.748]
  Call Extruder(14328.14707)
  MoveL 1459 to (-8.31, -10.42, 65) mm, rotated rx 180 ry 0 rz 180 deg; joints [-161.2, -56.679, -93.213, 21.481, 61.649, -10.585]
  Call Extruder(14332.81071)
  MoveL 1460 to (-5.78, -12.01, 65) mm, rotated rx 180 ry 0 rz 180 deg; joints [-161.572, -56.773, -92.893, 21.11, 61.37, -10.48]
  Call Extruder(14337.47427)
  MoveL 1461 to (-2.97, -13, 65) mm, rotated rx -180 ry 0 rz 180 deg; joints [-161.863, -56.891, -92.491, 20.839, 61.053, -10.439]
  Call Extruder(14342.17269)
  MoveL 1462 to (0.02, -13.33, 65) mm, rotated rx 180 ry 0 rz -180 deg; joints [-162.06, -57.03, -92.024, 20.682, 60.71, -10.464]
  Set speed (130.0 mm/s)
  MoveL 1463 to (0.02, -13.33, 70) mm, rotated rx 180 ry 0 rz -180 deg; joints [-162.06, -56.261, -92.4, 20.76, 60.343, -10.623]
  MoveL 1464 to (-26.25, -4.54, 70) mm, rotated rx 180 ry 0 rz -180 deg; joints [-159.288, -55.182, -96.089, 23.325, 63.282, -10.971]
  Call Extruder(14344.40532)
  Set speed (60.0 mm/s)
  MoveL 1465 to (-26.09, -5.96, 70) mm, rotated rx 180 ry 0 rz 180 deg; joints [-159.522, -55.166, -96.147, 23.06, 63.276, -10.837]
  Call Extruder(14353.77011)
  MoveL 1466 to (-24.12, -11.61, 70) mm, rotated rx 180 ry 0 rz 180 deg; joints [-160.532, -55.162, -96.159, 21.946, 63.099, -10.332]
  Call Extruder(14363.13503)
  MoveL 1467 to (-20.93, -16.69, 70) mm, rotated rx 180 ry 0 rz 180 deg; joints [-161.513, -55.225, -95.933, 20.891, 62.774, -9.905]
  Call Extruder(14372.50024)
  MoveL 1468 to (-16.69, -20.93, 70) mm, rotated rx -180 ry 0 rz 180 deg; joints [-162.406, -55.353, -95.481, 19.958, 62.319, -9.576]
  Call Extruder(14381.86516)
  MoveL 1469 to (-11.61, -24.12, 70) mm, rotated rx 180 ry 0 rz 180 deg; joints [-163.159, -55.539, -94.828, 19.2, 61.756, -9.358]
  Call Extruder(14391.22995)
  MoveL 1470 to (-5.96, -26.09, 70) mm, rotated rx -180 ry 0 rz -180 deg; joints [-163.733, -55.778, -94.01, 18.658, 61.115, -9.264]
  Call Extruder(14400.59505)
  MoveL 1471 to (0, -26.77, 70) mm, rotated rx -180 ry 0 rz 180 deg; joints [-164.103, -56.058, -93.072, 18.356, 60.43, -9.299]
  Call Extruder(14403.63717)
  MoveL 1472 to (1.93, -26.55, 70) mm, rotated rx 180 ry 0 rz 180 deg; joints [-164.154, -56.157, -92.744, 18.339, 60.205, -9.353]
  Call Extruder(14409.96016)
  MoveL 1473 to (5.96, -26.09, 70) mm, rotated rx 180 ry 0 rz -180 deg; joints [-164.258, -56.366, -92.061, 18.307, 59.738, -9.466]
  Call Extruder(14419.32496)
  MoveL 1474 to (11.61, -24.11, 70) mm, rotated rx 180 ry 0 rz 180 deg; joints [-164.201, -56.687, -91.029, 18.505, 59.073, -9.76]
  Call Extruder(14428.68987)
  MoveL 1475 to (16.69, -20.93, 70) mm, rotated rx 180 ry 0 rz 180 deg; joints [-163.944, -57.006, -90.027, 18.934, 58.471, -10.17]
  Call Extruder(14438.05508)
  MoveL 1476 to (20.93, -16.69, 70) mm, rotated rx 180 ry 0 rz 180 deg; joints [-163.508, -57.305, -89.104, 19.566, 57.961, -10.678]
  Call Extruder(14447.42000)
  MoveL 1477 to (24.12, -11.61, 70) mm, rotated rx 180 ry 0 rz 180 deg; joints [-162.92, -57.568, -88.305, 20.364, 57.569, -11.258]
  Call Extruder(14456.78479)
  MoveL 1478 to (26.09, -5.96, 70) mm, rotated rx 180 ry 0 rz -180 deg; joints [-162.209, -57.78, -87.667, 21.286, 57.314, -11.882]
  Call Extruder(14466.14990)
  MoveL 1479 to (26.77, 0, 70) mm, rotated rx 180 ry 0 rz -180 deg; joints [-161.41, -57.931, -87.22, 22.286, 57.207, -12.515]
  Call Extruder(14475.51500)
  MoveL 1480 to (26.09, 5.96, 70) mm, rotated rx -180 ry 0 rz -180 deg; joints [-160.556, -58.01, -86.986, 23.315, 57.254, -13.123]
  Call Extruder(14484.87980)
  MoveL 1481 to (24.12, 11.61, 70) mm, rotated rx 180 ry 0 rz 180 deg; joints [-159.683, -58.014, -86.975, 24.326, 57.449, -13.67]
  Call Extruder(14494.24472)
  MoveL 1482 to (20.93, 16.69, 70) mm, rotated rx 180 ry 0 rz 180 deg; joints [-158.826, -57.942, -87.187, 25.274, 57.783, -14.128]
  Call Extruder(14503.60992)
  MoveL 1483 to (16.69, 20.93, 70) mm, rotated rx 180 ry 0 rz 180 deg; joints [-158.019, -57.798, -87.614, 26.118, 58.237, -14.472]
  Call Extruder(14512.97483)
  MoveL 1484 to (11.61, 24.11, 70) mm, rotated rx 180 ry 0 rz 180 deg; joints [-157.299, -57.591, -88.234, 26.823, 58.788, -14.683]
  Call Extruder(14522.33964)
  MoveL 1485 to (5.96, 26.09, 70) mm, rotated rx 180 ry 0 rz -180 deg; joints [-156.697, -57.333, -89.019, 27.358, 59.41, -14.752]
  Call Extruder(14531.70474)
  MoveL 1486 to (0, 26.77, 70) mm, rotated rx 180 ry 0 rz 180 deg; joints [-156.245, -57.037, -89.931, 27.698, 60.071, -14.677]
  Call Extruder(14541.06984)
  MoveL 1487 to (-5.96, 26.09, 70) mm, rotated rx 180 ry 0 rz -180 deg; joints [-155.969, -56.719, -90.927, 27.826, 60.741, -14.465]
  Call Extruder(14550.43464)
  MoveL 1488 to (-11.61, 24.11, 70) mm, rotated rx 180 ry 0 rz 180 deg; joints [-155.891, -56.397, -91.958, 27.729, 61.387, -14.13]
  Call Extruder(14559.79956)
  MoveL 1489 to (-16.69, 20.93, 70) mm, rotated rx -180 ry 0 rz -180 deg; joints [-156.025, -56.087, -92.974, 27.406, 61.981, -13.689]
  Call Extruder(14569.16476)
  MoveL 1490 to (-20.93, 16.69, 70) mm, rotated rx 180 ry 0 rz 180 deg; joints [-156.374, -55.804, -93.922, 26.863, 62.491, -13.168]
  Call Extruder(14578.52968)
  MoveL 1491 to (-24.11, 11.61, 70) mm, rotated rx 180 ry 0 rz 180 deg; joints [-156.928, -55.561, -94.754, 26.119, 62.895, -12.593]
  Call Extruder(14587.89448)
  MoveL 1492 to (-26.09, 5.96, 70) mm, rotated rx -180 ry 0 rz 180 deg; joints [-157.665, -55.369, -95.424, 25.206, 63.169, -11.994]
  Call Extruder(14597.25958)
  MoveL 1493 to (-26.77, 0, 70) mm, rotated rx 180 ry 0 rz -180 deg; joints [-158.546, -55.235, -95.898, 24.168, 63.3, -11.4]
  Call Extruder(14602.04831)
  MoveL 1494 to (-26.42, -3.05, 70) mm, rotated rx 180 ry 0 rz 180 deg; joints [-159.044, -55.199, -96.027, 23.602, 63.288, -11.112]
  Set speed (130.0 mm/s)
  MoveL 1495 to (-41.86, -6.29, 70) mm, rotated rx 180 ry 0 rz 180 deg; joints [-158.606, -54.513, -98.583, 23.718, 65.082, -10.487]
  Call Extruder(14607.04616)
  Set speed (60.0 mm/s)
  MoveL 1496 to (-41.51, -9.47, 70) mm, rotated rx 180 ry 0 rz 180 deg; joints [-159.151, -54.479, -98.715, 23.107, 65.074, -10.194]
  Call Extruder(14621.94181)
  MoveL 1497 to (-38.36, -18.47, 70) mm, rotated rx 180 ry 0 rz 180 deg; joints [-160.835, -54.474, -98.734, 21.273, 64.801, -9.412]
  Call Extruder(14636.83766)
  MoveL 1498 to (-33.29, -26.54, 70) mm, rotated rx 180 ry 0 rz 180 deg; joints [-162.466, -54.569, -98.365, 19.535, 64.287, -8.752]
  Call Extruder(14651.73348)
  MoveL 1499 to (-26.54, -33.28, 70) mm, rotated rx 180 ry 0 rz -180 deg; joints [-163.93, -54.762, -97.63, 18.009, 63.557, -8.237]
  Call Extruder(14666.62934)
  MoveL 1500 to (-18.47, -38.36, 70) mm, rotated rx 180 ry 0 rz 180 deg; joints [-165.137, -55.048, -96.574, 16.786, 62.652, -7.889]
  Call Extruder(14681.52498)
  MoveL 1501 to (-9.47, -41.5, 70) mm, rotated rx 180 ry 0 rz 180 deg; joints [-166.024, -55.417, -95.256, 15.932, 61.621, -7.727]
  Call Extruder(14696.42086)
  MoveL 1502 to (0, -42.57, 70) mm, rotated rx 180 ry 0 rz 180 deg; joints [-166.562, -55.854, -93.751, 15.483, 60.522, -7.762]
  Call Extruder(14702.22851)
  MoveL 1503 to (3.69, -42.16, 70) mm, rotated rx 180 ry 0 rz 180 deg; joints [-166.635, -56.041, -93.125, 15.467, 60.088, -7.856]
  Call Extruder(14711.31673)
  MoveL 1504 to (9.47, -41.51, 70) mm, rotated rx 180 ry 0 rz 180 deg; joints [-166.745, -56.342, -92.138, 15.447, 59.412, -8.004]
  Call Extruder(14726.21239)
  MoveL 1505 to (18.47, -38.36, 70) mm, rotated rx -180 ry 0 rz 180 deg; joints [-166.591, -56.855, -90.499, 15.808, 58.349, -8.45]
  Call Extruder(14741.10824)
  MoveL 1506 to (26.54, -33.28, 70) mm, rotated rx 180 ry 0 rz 180 deg; joints [-166.133, -57.367, -88.914, 16.531, 57.389, -9.088]
  Call Extruder(14756.00406)
  MoveL 1507 to (33.28, -26.54, 70) mm, rotated rx -180 ry 0 rz 180 deg; joints [-165.409, -57.85, -87.459, 17.567, 56.578, -9.891]
  Call Extruder(14770.89991)
  MoveL 1508 to (38.36, -18.47, 70) mm, rotated rx -180 ry 0 rz -180 deg; joints [-164.468, -58.278, -86.201, 18.854, 55.958, -10.822]
  Call Extruder(14785.79556)
  MoveL 1509 to (41.5, -9.47, 70) mm, rotated rx 180 ry 0 rz 180 deg; joints [-163.355, -58.624, -85.198, 20.324, 55.559, -11.831]
  Call Extruder(14800.69144)
  MoveL 1510 to (42.57, 0, 70) mm, rotated rx -180 ry 0 rz 180 deg; joints [-162.12, -58.87, -84.496, 21.901, 55.397, -12.86]
  Call Extruder(14815.58731)
  MoveL 1511 to (41.51, 9.47, 70) mm, rotated rx 180 ry 0 rz 180 deg; joints [-160.81, -58.999, -84.128, 23.512, 55.48, -13.85]
  Call Extruder(14830.48297)
  MoveL 1512 to (38.36, 18.47, 70) mm, rotated rx 180 ry 0 rz 180 deg; joints [-159.475, -59.006, -84.111, 25.083, 55.799, -14.74]
  Call Extruder(14845.37882)
  MoveL 1513 to (33.28, 26.54, 70) mm, rotated rx 180 ry 0 rz 180 deg; joints [-158.16, -58.888, -84.444, 26.549, 56.336, -15.481]
  Call Extruder(14860.27464)
  MoveL 1514 to (26.54, 33.28, 70) mm, rotated rx -180 ry 0 rz 180 deg; joints [-156.916, -58.653, -85.114, 27.851, 57.061, -16.03]
  Call Extruder(14875.17048)
  MoveL 1515 to (18.47, 38.36, 70) mm, rotated rx 180 ry 0 rz -180 deg; joints [-155.789, -58.316, -86.089, 28.942, 57.937, -16.36]
  Call Extruder(14890.06615)
  MoveL 1516 to (9.47, 41.51, 70) mm, rotated rx -180 ry 0 rz 180 deg; joints [-154.828, -57.896, -87.324, 29.778, 58.918, -16.457]
  Call Extruder(14904.96202)
  MoveL 1517 to (0, 42.57, 70) mm, rotated rx 180 ry 0 rz 180 deg; joints [-154.081, -57.417, -88.763, 30.326, 59.96, -16.322]
  Call Extruder(14919.85789)
  MoveL 1518 to (-9.47, 41.51, 70) mm, rotated rx 180 ry 0 rz 180 deg; joints [-153.594, -56.906, -90.338, 30.558, 61.013, -15.967]
  Call Extruder(14934.75354)
  MoveL 1519 to (-18.47, 38.36, 70) mm, rotated rx 180 ry 0 rz -180 deg; joints [-153.408, -56.392, -91.976, 30.452, 62.031, -15.415]
  Call Extruder(14949.64939)
  MoveL 1520 to (-26.54, 33.28, 70) mm, rotated rx -180 ry 0 rz 180 deg; joints [-153.557, -55.901, -93.595, 29.995, 62.967, -14.7]
  Call Extruder(14964.54521)
  MoveL 1521 to (-33.28, 26.54, 70) mm, rotated rx 180 ry 0 rz -180 deg; joints [-154.059, -55.457, -95.114, 29.184, 63.779, -13.862]
  Call Extruder(14979.44106)
  MoveL 1522 to (-38.36, 18.47, 70) mm, rotated rx 180 ry 0 rz 180 deg; joints [-154.913, -55.081, -96.453, 28.037, 64.426, -12.946]
  Call Extruder(14994.33672)
  MoveL 1523 to (-41.5, 9.47, 70) mm, rotated rx 180 ry 0 rz -180 deg; joints [-156.091, -54.786, -97.539, 26.593, 64.875, -12]
  Call Extruder(15009.23260)
  MoveL 1524 to (-42.57, 0, 70) mm, rotated rx 180 ry 0 rz -180 deg; joints [-157.533, -54.584, -98.308, 24.918, 65.097, -11.069]
  Call Extruder(15016.78687)
  MoveL 1525 to (-42.03, -4.8, 70) mm, rotated rx 180 ry 0 rz 180 deg; joints [-158.35, -54.529, -98.52, 24.003, 65.086, -10.624]
  Set speed (130.0 mm/s)
  MoveL 1526 to (-54.1, -7.67, 70) mm, rotated rx 180 ry 0 rz 180 deg; joints [-158.024, -54.038, -100.496, 24.083, 66.501, -10.105]
  Call Extruder(15020.85950)
  Set speed (30.0 mm/s)
  MoveL 1527 to (-53.59, -12.23, 70) mm, rotated rx 180 ry 0 rz 180 deg; joints [-158.835, -53.992, -100.687, 23.186, 66.495, -9.694]
  Call Extruder(15031.78963)
  MoveL 1528 to (-49.52, -23.85, 70) mm, rotated rx -180 ry 0 rz 180 deg; joints [-161.095, -53.986, -100.713, 20.747, 66.151, -8.708]
  Call Extruder(15042.71992)
  MoveL 1529 to (-42.98, -34.27, 70) mm, rotated rx -180 ry 0 rz 180 deg; joints [-163.275, -54.102, -100.226, 18.438, 65.488, -7.875]
  Call Extruder(15053.65004)
  MoveL 1530 to (-34.27, -42.98, 70) mm, rotated rx 180 ry 0 rz 180 deg; joints [-165.21, -54.341, -99.26, 16.423, 64.539, -7.222]
  Call Extruder(15064.58032)
  MoveL 1531 to (-23.85, -49.53, 70) mm, rotated rx 180 ry 0 rz 180 deg; joints [-166.774, -54.697, -97.876, 14.831, 63.359, -6.771]
  Call Extruder(15075.51045)
  MoveL 1532 to (-12.23, -53.59, 70) mm, rotated rx 180 ry 0 rz 180 deg; joints [-167.889, -55.163, -96.157, 13.744, 62.015, -6.547]
  Call Extruder(15086.44068)
  MoveL 1533 to (0, -54.97, 70) mm, rotated rx 180 ry 0 rz 180 deg; joints [-168.526, -55.721, -94.203, 13.2, 60.585, -6.571]
  Call Extruder(15090.97367)
  MoveL 1534 to (5.07, -54.4, 70) mm, rotated rx -180 ry 0 rz 180 deg; joints [-168.599, -55.976, -93.342, 13.197, 59.987, -6.69]
  Call Extruder(15097.37090)
  MoveL 1535 to (12.23, -53.59, 70) mm, rotated rx -180 ry 0 rz 180 deg; joints [-168.697, -56.348, -92.117, 13.198, 59.145, -6.858]
  Call Extruder(15108.30104)
  MoveL 1536 to (23.85, -49.53, 70) mm, rotated rx -180 ry 0 rz 180 deg; joints [-168.436, -57.013, -90.004, 13.708, 57.769, -7.412]
  Call Extruder(15119.23132)
  MoveL 1537 to (34.27, -42.98, 70) mm, rotated rx -180 ry 0 rz 180 deg; joints [-167.797, -57.68, -87.967, 14.679, 56.527, -8.221]
  Call Extruder(15130.16144)
  MoveL 1538 to (42.98, -34.27, 70) mm, rotated rx 180 ry 0 rz 180 deg; joints [-166.837, -58.312, -86.099, 16.044, 55.482, -9.256]
  Call Extruder(15141.09172)
  MoveL 1539 to (49.53, -23.85, 70) mm, rotated rx 180 ry 0 rz 180 deg; joints [-165.618, -58.873, -84.487, 17.722, 54.684, -10.467]
  Call Extruder(15152.02186)
  MoveL 1540 to (53.59, -12.23, 70) mm, rotated rx 180 ry 0 rz -180 deg; joints [-164.2, -59.329, -83.202, 19.623, 54.172, -11.788]
  Call Extruder(15162.95208)
  MoveL 1541 to (54.97, 0, 70) mm, rotated rx -180 ry 0 rz 180 deg; joints [-162.641, -59.652, -82.304, 21.65, 53.971, -13.142]
  Call Extruder(15173.88230)
  MoveL 1542 to (53.59, 12.23, 70) mm, rotated rx 180 ry 0 rz 180 deg; joints [-160.996, -59.823, -81.833, 23.707, 54.086, -14.444]
  Call Extruder(15184.81244)
  MoveL 1543 to (49.52, 23.85, 70) mm, rotated rx -180 ry 0 rz -180 deg; joints [-159.322, -59.831, -81.81, 25.703, 54.507, -15.613]
  Call Extruder(15195.74272)
  MoveL 1544 to (42.98, 34.27, 70) mm, rotated rx -180 ry 0 rz 180 deg; joints [-157.673, -59.676, -82.238, 27.555, 55.208, -16.58]
  Call Extruder(15206.67284)
  MoveL 1545 to (34.27, 42.98, 70) mm, rotated rx 180 ry 0 rz 180 deg; joints [-156.102, -59.367, -83.095, 29.196, 56.148, -17.29]
  Call Extruder(15217.60312)
  MoveL 1546 to (23.85, 49.52, 70) mm, rotated rx -180 ry 0 rz 180 deg; joints [-154.667, -58.923, -84.343, 30.57, 57.277, -17.709]
  Call Extruder(15228.53326)
  MoveL 1547 to (12.23, 53.59, 70) mm, rotated rx -180 ry 0 rz 180 deg; joints [-153.426, -58.372, -85.926, 31.631, 58.539, -17.821]
  Call Extruder(15239.46348)
  MoveL 1548 to (0, 54.97, 70) mm, rotated rx -180 ry 0 rz -180 deg; joints [-152.438, -57.745, -87.773, 32.342, 59.874, -17.63]
  Call Extruder(15250.39371)
  MoveL 1549 to (-12.23, 53.59, 70) mm, rotated rx 180 ry 0 rz 180 deg; joints [-151.764, -57.08, -89.797, 32.668, 61.222, -17.155]
  Call Extruder(15261.32384)
  MoveL 1550 to (-23.85, 49.52, 70) mm, rotated rx 180 ry 0 rz 180 deg; joints [-151.463, -56.413, -91.907, 32.579, 62.524, -16.426]
  Call Extruder(15272.25412)
  MoveL 1551 to (-34.27, 42.98, 70) mm, rotated rx 180 ry 0 rz 180 deg; joints [-151.589, -55.781, -94, 32.047, 63.724, -15.49]
  Call Extruder(15283.18424)
  MoveL 1552 to (-42.98, 34.27, 70) mm, rotated rx -180 ry 0 rz -180 deg; joints [-152.179, -55.214, -95.972, 31.059, 64.77, -14.398]
  Call Extruder(15294.11452)
  MoveL 1553 to (-49.52, 23.85, 70) mm, rotated rx 180 ry 0 rz 180 deg; joints [-153.248, -54.739, -97.719, 29.619, 65.612, -13.211]
  Call Extruder(15305.04466)
  MoveL 1554 to (-53.59, 12.23, 70) mm, rotated rx 180 ry 0 rz 180 deg; joints [-154.769, -54.371, -99.14, 27.766, 66.204, -11.993]
  Call Extruder(15315.97488)
  MoveL 1555 to (-54.97, 0, 70) mm, rotated rx 180 ry 0 rz -180 deg; joints [-156.673, -54.121, -100.151, 25.58, 66.508, -10.803]
  Call Extruder(15321.50050)
  MoveL 1556 to (-54.27, -6.18, 70) mm, rotated rx 180 ry 0 rz -180 deg; joints [-157.76, -54.053, -100.432, 24.375, 66.503, -10.24]
  Set speed (130.0 mm/s)
  MoveL 1557 to (-49.9, -9.51, 70) mm, rotated rx 180 ry 0 rz -180 deg; joints [-158.616, -54.162, -99.98, 23.515, 66.039, -10.022]
  MoveL 1558 to (0.44, -13.28, 70) mm, rotated rx 180 ry 0 rz 180 deg; joints [-162.073, -56.283, -92.33, 20.755, 60.295, -10.636]
  Call Extruder(15325.47307)
  Set speed (80.0 mm/s)
  MoveL 1559 to (2.97, -12.99, 70) mm, rotated rx -180 ry 0 rz -180 deg; joints [-162.152, -56.415, -91.902, 20.725, 60.003, -10.712]
  Call Extruder(15330.13663)
  MoveL 1560 to (5.78, -12.01, 70) mm, rotated rx 180 ry 0 rz 180 deg; joints [-162.141, -56.575, -91.388, 20.812, 59.674, -10.864]
  Call Extruder(15334.80025)
  MoveL 1561 to (8.31, -10.42, 70) mm, rotated rx -180 ry 0 rz -180 deg; joints [-162.027, -56.732, -90.887, 21.013, 59.375, -11.072]
  Call Extruder(15339.46445)
  MoveL 1562 to (10.42, -8.31, 70) mm, rotated rx -180 ry 0 rz -180 deg; joints [-161.819, -56.879, -90.424, 21.319, 59.121, -11.326]
  Call Extruder(15344.12808)
  MoveL 1563 to (12.01, -5.78, 70) mm, rotated rx 180 ry 0 rz 180 deg; joints [-161.529, -57.007, -90.022, 21.711, 58.924, -11.614]
  Call Extruder(15348.79165)
  MoveL 1564 to (13, -2.97, 70) mm, rotated rx 180 ry 0 rz -180 deg; joints [-161.171, -57.111, -89.701, 22.169, 58.795, -11.92]
  Call Extruder(15353.45560)
  MoveL 1565 to (13.33, 0, 70) mm, rotated rx 180 ry 0 rz 180 deg; joints [-160.763, -57.184, -89.476, 22.671, 58.74, -12.23]
  Call Extruder(15358.11955)
  MoveL 1566 to (12.99, 2.97, 70) mm, rotated rx 180 ry 0 rz 180 deg; joints [-160.324, -57.222, -89.357, 23.191, 58.761, -12.527]
  Call Extruder(15362.78313)
  MoveL 1567 to (12.01, 5.78, 70) mm, rotated rx 180 ry 0 rz -180 deg; joints [-159.874, -57.224, -89.352, 23.706, 58.856, -12.795]
  Call Extruder(15367.44675)
  MoveL 1568 to (10.42, 8.31, 70) mm, rotated rx 180 ry 0 rz 180 deg; joints [-159.432, -57.189, -89.459, 24.19, 59.02, -13.019]
  Call Extruder(15372.11094)
  MoveL 1569 to (8.31, 10.42, 70) mm, rotated rx 180 ry 0 rz 180 deg; joints [-159.021, -57.12, -89.674, 24.621, 59.246, -13.189]
  Call Extruder(15376.77457)
  MoveL 1570 to (5.78, 12.01, 70) mm, rotated rx 180 ry 0 rz 180 deg; joints [-158.657, -57.019, -89.987, 24.98, 59.522, -13.295]
  Call Extruder(15381.43814)
  MoveL 1571 to (2.97, 13, 70) mm, rotated rx 180 ry 0 rz 180 deg; joints [-158.359, -56.892, -90.381, 25.249, 59.833, -13.333]
  Call Extruder(15386.10209)
  MoveL 1572 to (0, 13.33, 70) mm, rotated rx 180 ry 0 rz 180 deg; joints [-158.143, -56.747, -90.839, 25.415, 60.165, -13.3]
  Call Extruder(15390.76605)
  MoveL 1573 to (-2.97, 13, 70) mm, rotated rx 180 ry 0 rz 180 deg; joints [-158.019, -56.59, -91.337, 25.47, 60.502, -13.2]
  Call Extruder(15395.42961)
  MoveL 1574 to (-5.78, 12.01, 70) mm, rotated rx 180 ry 0 rz -180 deg; joints [-157.997, -56.43, -91.851, 25.409, 60.827, -13.038]
  Call Extruder(15400.09324)
  MoveL 1575 to (-8.31, 10.42, 70) mm, rotated rx -180 ry 0 rz 180 deg; joints [-158.08, -56.275, -92.355, 25.234, 61.124, -12.822]
  Call Extruder(15404.75744)
  MoveL 1576 to (-10.42, 8.31, 70) mm, rotated rx 180 ry 0 rz 180 deg; joints [-158.266, -56.132, -92.824, 24.951, 61.378, -12.564]
  Call Extruder(15409.42106)
  MoveL 1577 to (-12.01, 5.78, 70) mm, rotated rx 180 ry 0 rz 180 deg; joints [-158.549, -56.009, -93.234, 24.572, 61.577, -12.278]
  Call Extruder(15414.08463)
  MoveL 1578 to (-12.99, 2.97, 70) mm, rotated rx 180 ry 0 rz -180 deg; joints [-158.913, -55.91, -93.564, 24.116, 61.711, -11.978]
  Call Extruder(15418.74859)
  MoveL 1579 to (-13.33, 0, 70) mm, rotated rx -180 ry 0 rz 180 deg; joints [-159.341, -55.841, -93.796, 23.604, 61.772, -11.677]
  Call Extruder(15423.41254)
  MoveL 1580 to (-12.99, -2.97, 70) mm, rotated rx 180 ry 0 rz 180 deg; joints [-159.811, -55.805, -93.918, 23.064, 61.757, -11.392]
  Call Extruder(15428.07611)
  MoveL 1581 to (-12.01, -5.78, 70) mm, rotated rx -180 ry 0 rz 180 deg; joints [-160.294, -55.803, -93.923, 22.524, 61.667, -11.135]
  Call Extruder(15432.73973)
  MoveL 1582 to (-10.42, -8.31, 70) mm, rotated rx 180 ry 0 rz 180 deg; joints [-160.766, -55.836, -93.813, 22.014, 61.504, -10.918]
  Call Extruder(15437.40392)
  MoveL 1583 to (-8.31, -10.42, 70) mm, rotated rx 180 ry 0 rz 180 deg; joints [-161.2, -55.902, -93.591, 21.561, 61.278, -10.751]
  Call Extruder(15442.06756)
  MoveL 1584 to (-5.78, -12.01, 70) mm, rotated rx 180 ry 0 rz 180 deg; joints [-161.572, -55.998, -93.271, 21.189, 61, -10.644]
  Call Extruder(15446.73112)
  MoveL 1585 to (-2.97, -12.99, 70) mm, rotated rx 180 ry 0 rz -180 deg; joints [-161.863, -56.119, -92.868, 20.917, 60.684, -10.6]
  Call Extruder(15451.39506)
  MoveL 1586 to (0, -13.33, 70) mm, rotated rx 180 ry 0 rz -180 deg; joints [-162.059, -56.26, -92.404, 20.761, 60.346, -10.623]
  Call Extruder(15452.08647)
  MoveL 1587 to (0.44, -13.28, 70) mm, rotated rx 180 ry 0 rz 180 deg; joints [-162.073, -56.283, -92.33, 20.755, 60.295, -10.636]
  Set speed (130.0 mm/s)
  MoveL 1588 to (0.44, -13.28, 75) mm, rotated rx 180 ry 0 rz 180 deg; joints [-162.073, -55.515, -92.697, 20.837, 59.92, -10.8]
  MoveL 1589 to (-26.25, -4.54, 75) mm, rotated rx 180 ry 0 rz 180 deg; joints [-159.288, -54.386, -96.464, 23.409, 62.896, -11.158]
  Call Extruder(15454.31909)
  Set speed (60.0 mm/s)
  MoveL 1590 to (-26.09, -5.96, 75) mm, rotated rx -180 ry 0 rz 180 deg; joints [-159.522, -54.37, -96.522, 23.144, 62.889, -11.023]
  Call Extruder(15463.68388)
  MoveL 1591 to (-24.12, -11.61, 75) mm, rotated rx -180 ry 0 rz 180 deg; joints [-160.532, -54.366, -96.534, 22.027, 62.708, -10.509]
  Call Extruder(15473.04880)
  MoveL 1592 to (-20.93, -16.69, 75) mm, rotated rx 180 ry 0 rz 180 deg; joints [-161.513, -54.431, -96.307, 20.969, 62.382, -10.074]
  Call Extruder(15482.41401)
  MoveL 1593 to (-16.69, -20.93, 75) mm, rotated rx -180 ry 0 rz -180 deg; joints [-162.406, -54.562, -95.854, 20.034, 61.927, -9.737]
  Call Extruder(15491.77893)
  MoveL 1594 to (-11.61, -24.12, 75) mm, rotated rx 180 ry 0 rz 180 deg; joints [-163.159, -54.754, -95.2, 19.274, 61.365, -9.513]
  Call Extruder(15501.14372)
  MoveL 1595 to (-5.96, -26.09, 75) mm, rotated rx 180 ry 0 rz -180 deg; joints [-163.733, -54.998, -94.381, 18.731, 60.727, -9.414]
  Call Extruder(15510.50882)
  MoveL 1596 to (0, -26.77, 75) mm, rotated rx 180 ry 0 rz 180 deg; joints [-164.103, -55.284, -93.44, 18.429, 60.046, -9.446]
  Call Extruder(15514.20698)
  MoveL 1597 to (2.35, -26.5, 75) mm, rotated rx -180 ry 0 rz -180 deg; joints [-164.165, -55.407, -93.041, 18.409, 59.775, -9.512]
  Call Extruder(15519.87393)
  MoveL 1598 to (5.96, -26.09, 75) mm, rotated rx 180 ry 0 rz 180 deg; joints [-164.258, -55.599, -92.427, 18.381, 59.359, -9.612]
  Call Extruder(15529.23873)
  MoveL 1599 to (11.61, -24.11, 75) mm, rotated rx 180 ry 0 rz 180 deg; joints [-164.201, -55.928, -91.394, 18.581, 58.699, -9.907]
  Call Extruder(15538.60364)
  MoveL 1600 to (16.69, -20.93, 75) mm, rotated rx 180 ry 0 rz 180 deg; joints [-163.944, -56.253, -90.39, 19.013, 58.103, -10.319]
  Call Extruder(15547.96885)
  MoveL 1601 to (20.93, -16.69, 75) mm, rotated rx 180 ry 0 rz 180 deg; joints [-163.508, -56.558, -89.467, 19.647, 57.598, -10.83]
  Call Extruder(15557.33377)
  MoveL 1602 to (24.11, -11.61, 75) mm, rotated rx -180 ry 0 rz 180 deg; joints [-162.92, -56.825, -88.666, 20.449, 57.212, -11.416]
  Call Extruder(15566.69856)
  MoveL 1603 to (26.09, -5.96, 75) mm, rotated rx 180 ry 0 rz -180 deg; joints [-162.209, -57.042, -88.028, 21.375, 56.961, -12.046]
  Call Extruder(15576.06366)
  MoveL 1604 to (26.77, 0, 75) mm, rotated rx 180 ry 0 rz -180 deg; joints [-161.41, -57.195, -87.58, 22.378, 56.859, -12.685]
  Call Extruder(15585.42877)
  MoveL 1605 to (26.09, 5.96, 75) mm, rotated rx -180 ry 0 rz 180 deg; joints [-160.556, -57.275, -87.346, 23.411, 56.91, -13.3]
  Call Extruder(15594.79357)
  MoveL 1606 to (24.11, 11.61, 75) mm, rotated rx -180 ry 0 rz 180 deg; joints [-159.683, -57.279, -87.335, 24.425, 57.108, -13.854]
  Call Extruder(15604.15848)
  MoveL 1607 to (20.93, 16.69, 75) mm, rotated rx 180 ry 0 rz 180 deg; joints [-158.826, -57.206, -87.547, 25.376, 57.443, -14.319]
  Call Extruder(15613.52369)
  MoveL 1608 to (16.69, 20.93, 75) mm, rotated rx -180 ry 0 rz 180 deg; joints [-158.019, -57.06, -87.974, 26.222, 57.898, -14.668]
  Call Extruder(15622.88861)
  MoveL 1609 to (11.61, 24.11, 75) mm, rotated rx 180 ry 0 rz 180 deg; joints [-157.299, -56.849, -88.595, 26.928, 58.449, -14.884]
  Call Extruder(15632.25341)
  MoveL 1610 to (5.96, 26.09, 75) mm, rotated rx 180 ry 0 rz 180 deg; joints [-156.697, -56.586, -89.381, 27.463, 59.068, -14.958]
  Call Extruder(15641.61851)
  MoveL 1611 to (0, 26.77, 75) mm, rotated rx -180 ry 0 rz 180 deg; joints [-156.245, -56.284, -90.294, 27.803, 59.727, -14.887]
  Call Extruder(15650.98361)
  MoveL 1612 to (-5.96, 26.09, 75) mm, rotated rx 180 ry 0 rz 180 deg; joints [-155.969, -55.96, -91.292, 27.93, 60.393, -14.677]
  Call Extruder(15660.34841)
  MoveL 1613 to (-11.61, 24.12, 75) mm, rotated rx 180 ry 0 rz 180 deg; joints [-155.891, -55.632, -92.325, 27.831, 61.034, -14.342]
  Call Extruder(15669.71333)
  MoveL 1614 to (-16.69, 20.93, 75) mm, rotated rx 180 ry 0 rz -180 deg; joints [-156.025, -55.314, -93.342, 27.506, 61.622, -13.9]
  Call Extruder(15679.07853)
  MoveL 1615 to (-20.93, 16.69, 75) mm, rotated rx 180 ry 0 rz 180 deg; joints [-156.374, -55.025, -94.292, 26.96, 62.127, -13.377]
  Call Extruder(15688.44345)
  MoveL 1616 to (-24.11, 11.61, 75) mm, rotated rx 180 ry 0 rz 180 deg; joints [-156.928, -54.776, -95.125, 26.213, 62.524, -12.798]
  Call Extruder(15697.80825)
  MoveL 1617 to (-26.09, 5.96, 75) mm, rotated rx -180 ry 0 rz 180 deg; joints [-157.665, -54.578, -95.798, 25.297, 62.792, -12.194]
  Call Extruder(15707.17335)
  MoveL 1618 to (-26.77, 0, 75) mm, rotated rx 180 ry 0 rz 180 deg; joints [-158.546, -54.441, -96.272, 24.255, 62.917, -11.593]
  Call Extruder(15711.96208)
  MoveL 1619 to (-26.42, -3.05, 75) mm, rotated rx -180 ry 0 rz 180 deg; joints [-159.044, -54.404, -96.402, 23.688, 62.903, -11.301]
  Set speed (130.0 mm/s)
  MoveL 1620 to (-41.86, -6.29, 75) mm, rotated rx 180 ry 0 rz 180 deg; joints [-158.606, -53.698, -98.964, 23.8, 64.685, -10.68]
  Call Extruder(15716.95993)
  Set speed (60.0 mm/s)
  MoveL 1621 to (-41.51, -9.47, 75) mm, rotated rx 180 ry 0 rz 180 deg; joints [-159.151, -53.663, -99.096, 23.188, 64.674, -10.383]
  Call Extruder(15731.85558)
  MoveL 1622 to (-38.36, -18.47, 75) mm, rotated rx -180 ry 0 rz 180 deg; joints [-160.835, -53.658, -99.115, 21.348, 64.395, -9.587]
  Call Extruder(15746.75144)
  MoveL 1623 to (-33.28, -26.54, 75) mm, rotated rx 180 ry 0 rz 180 deg; joints [-162.466, -53.756, -98.745, 19.606, 63.878, -8.913]
  Call Extruder(15761.64725)
  MoveL 1624 to (-26.54, -33.28, 75) mm, rotated rx -180 ry 0 rz -180 deg; joints [-163.93, -53.955, -98.009, 18.075, 63.149, -8.386]
  Call Extruder(15776.54311)
  MoveL 1625 to (-18.47, -38.36, 75) mm, rotated rx 180 ry 0 rz -180 deg; joints [-165.137, -54.249, -96.949, 16.849, 62.247, -8.028]
  Call Extruder(15791.43876)
  MoveL 1626 to (-9.47, -41.5, 75) mm, rotated rx 180 ry 0 rz 180 deg; joints [-166.024, -54.628, -95.629, 15.994, 61.221, -7.857]
  Call Extruder(15806.33463)
  MoveL 1627 to (0, -42.57, 75) mm, rotated rx 180 ry 0 rz 180 deg; joints [-166.562, -55.076, -94.121, 15.545, 60.128, -7.888]
  Call Extruder(15812.79833)
  MoveL 1628 to (4.11, -42.11, 75) mm, rotated rx 180 ry 0 rz 180 deg; joints [-166.643, -55.29, -93.423, 15.528, 59.65, -7.992]
  Call Extruder(15821.23051)
  MoveL 1629 to (9.47, -41.5, 75) mm, rotated rx 180 ry 0 rz 180 deg; joints [-166.745, -55.575, -92.505, 15.511, 59.026, -8.128]
  Call Extruder(15836.12617)
  MoveL 1630 to (18.47, -38.36, 75) mm, rotated rx -180 ry 0 rz 180 deg; joints [-166.591, -56.099, -90.864, 15.874, 57.972, -8.576]
  Call Extruder(15851.02201)
  MoveL 1631 to (26.54, -33.28, 75) mm, rotated rx 180 ry 0 rz 180 deg; joints [-166.133, -56.621, -89.276, 16.602, 57.021, -9.218]
  Call Extruder(15865.91783)
  MoveL 1632 to (33.28, -26.54, 75) mm, rotated rx 180 ry 0 rz 180 deg; joints [-165.409, -57.113, -87.819, 17.643, 56.219, -10.028]
  Call Extruder(15880.81368)
  MoveL 1633 to (38.36, -18.47, 75) mm, rotated rx -180 ry 0 rz 180 deg; joints [-164.468, -57.547, -86.56, 18.936, 55.607, -10.968]
  Call Extruder(15895.70934)
  MoveL 1634 to (41.5, -9.47, 75) mm, rotated rx -180 ry 0 rz 180 deg; joints [-163.355, -57.899, -85.556, 20.412, 55.215, -11.986]
  Call Extruder(15910.60521)
  MoveL 1635 to (42.57, 0, 75) mm, rotated rx -180 ry 0 rz 180 deg; joints [-162.12, -58.149, -84.854, 21.996, 55.06, -13.026]
  Call Extruder(15925.50108)
  MoveL 1636 to (41.5, 9.47, 75) mm, rotated rx 180 ry 0 rz 180 deg; joints [-160.81, -58.28, -84.486, 23.612, 55.148, -14.026]
  Call Extruder(15940.39675)
  MoveL 1637 to (38.36, 18.47, 75) mm, rotated rx 180 ry 0 rz 180 deg; joints [-159.475, -58.286, -84.468, 25.188, 55.472, -14.927]
  Call Extruder(15955.29259)
  MoveL 1638 to (33.29, 26.54, 75) mm, rotated rx 180 ry 0 rz 180 deg; joints [-158.16, -58.167, -84.802, 26.658, 56.012, -15.677]
  Call Extruder(15970.18841)
  MoveL 1639 to (26.54, 33.28, 75) mm, rotated rx -180 ry 0 rz 180 deg; joints [-156.916, -57.929, -85.472, 27.963, 56.738, -16.234]
  Call Extruder(15985.08425)
  MoveL 1640 to (18.47, 38.36, 75) mm, rotated rx 180 ry 0 rz -180 deg; joints [-155.789, -57.586, -86.448, 29.055, 57.612, -16.572]
  Call Extruder(15999.97992)
  MoveL 1641 to (9.47, 41.51, 75) mm, rotated rx 180 ry 0 rz 180 deg; joints [-154.828, -57.159, -87.684, 29.891, 58.592, -16.676]
  Call Extruder(16014.87579)
  MoveL 1642 to (0, 42.57, 75) mm, rotated rx 180 ry 0 rz 180 deg; joints [-154.081, -56.671, -89.125, 30.439, 59.629, -16.546]
  Call Extruder(16029.77167)
  MoveL 1643 to (-9.47, 41.51, 75) mm, rotated rx 180 ry 0 rz 180 deg; joints [-153.594, -56.151, -90.702, 30.669, 60.677, -16.195]
  Call Extruder(16044.66731)
  MoveL 1644 to (-18.47, 38.36, 75) mm, rotated rx -180 ry 0 rz -180 deg; joints [-153.408, -55.626, -92.342, 30.561, 61.687, -15.645]
  Call Extruder(16059.56317)
  MoveL 1645 to (-26.54, 33.28, 75) mm, rotated rx 180 ry 0 rz -180 deg; joints [-153.557, -55.124, -93.964, 30.1, 62.615, -14.93]
  Call Extruder(16074.45899)
  MoveL 1646 to (-33.29, 26.54, 75) mm, rotated rx -180 ry 0 rz 180 deg; joints [-154.059, -54.669, -95.487, 29.285, 63.416, -14.089]
  Call Extruder(16089.35483)
  MoveL 1647 to (-38.36, 18.47, 75) mm, rotated rx -180 ry 0 rz 180 deg; joints [-154.913, -54.283, -96.829, 28.133, 64.053, -13.167]
  Call Extruder(16104.25050)
  MoveL 1648 to (-41.5, 9.47, 75) mm, rotated rx 180 ry 0 rz 180 deg; joints [-156.091, -53.98, -97.917, 26.684, 64.492, -12.212]
  Call Extruder(16119.14637)
  MoveL 1649 to (-42.57, 0, 75) mm, rotated rx 180 ry 0 rz -180 deg; joints [-157.533, -53.771, -98.688, 25.004, 64.705, -11.27]
  Call Extruder(16126.70064)
  MoveL 1650 to (-42.03, -4.8, 75) mm, rotated rx 180 ry 0 rz -180 deg; joints [-158.35, -53.714, -98.9, 24.086, 64.69, -10.82]
  Set speed (130.0 mm/s)
  MoveL 1651 to (-54.1, -7.67, 75) mm, rotated rx 180 ry 0 rz 180 deg; joints [-158.024, -53.206, -100.882, 24.163, 66.094, -10.304]
  Call Extruder(16130.77328)
  Set speed (30.0 mm/s)
  MoveL 1652 to (-53.59, -12.23, 75) mm, rotated rx 180 ry 0 rz 180 deg; joints [-158.835, -53.159, -101.074, 23.264, 66.084, -9.887]
  Call Extruder(16141.70341)
  MoveL 1653 to (-49.52, -23.85, 75) mm, rotated rx 180 ry 0 rz 180 deg; joints [-161.095, -53.152, -101.1, 20.818, 65.734, -8.881]
  Call Extruder(16152.63369)
  MoveL 1654 to (-42.98, -34.27, 75) mm, rotated rx 180 ry 0 rz 180 deg; joints [-163.275, -53.273, -100.612, 18.503, 65.067, -8.03]
  Call Extruder(16163.56381)
  MoveL 1655 to (-34.27, -42.98, 75) mm, rotated rx 180 ry 0 rz 180 deg; joints [-165.21, -53.52, -99.643, 16.483, 64.119, -7.36]
  Call Extruder(16174.49409)
  MoveL 1656 to (-23.85, -49.53, 75) mm, rotated rx 180 ry 0 rz 180 deg; joints [-166.774, -53.888, -98.255, 14.887, 62.943, -6.895]
  Call Extruder(16185.42423)
  MoveL 1657 to (-12.23, -53.59, 75) mm, rotated rx 180 ry 0 rz 180 deg; joints [-167.889, -54.367, -96.532, 13.798, 61.607, -6.661]
  Call Extruder(16196.35445)
  MoveL 1658 to (0, -54.97, 75) mm, rotated rx 180 ry 0 rz 180 deg; joints [-168.526, -54.94, -94.574, 13.254, 60.185, -6.679]
  Call Extruder(16201.26028)
  MoveL 1659 to (5.49, -54.35, 75) mm, rotated rx 180 ry 0 rz 180 deg; joints [-168.604, -55.223, -93.64, 13.251, 59.543, -6.807]
  Call Extruder(16207.28467)
  MoveL 1660 to (12.23, -53.59, 75) mm, rotated rx 180 ry 0 rz 180 deg; joints [-168.697, -55.582, -92.484, 13.253, 58.755, -6.965]
  Call Extruder(16218.21481)
  MoveL 1661 to (23.85, -49.53, 75) mm, rotated rx 180 ry 0 rz 180 deg; joints [-168.436, -56.26, -90.368, 13.767, 57.391, -7.521]
  Call Extruder(16229.14509)
  MoveL 1662 to (34.27, -42.98, 75) mm, rotated rx 180 ry 0 rz 180 deg; joints [-167.797, -56.94, -88.328, 14.743, 56.16, -8.337]
  Call Extruder(16240.07521)
  MoveL 1663 to (42.98, -34.27, 75) mm, rotated rx -180 ry 0 rz 180 deg; joints [-166.837, -57.583, -86.458, 16.115, 55.125, -9.38]
  Call Extruder(16251.00549)
  MoveL 1664 to (49.53, -23.85, 75) mm, rotated rx -180 ry 0 rz 180 deg; joints [-165.618, -58.152, -84.844, 17.801, 54.338, -10.603]
  Call Extruder(16261.93563)
  MoveL 1665 to (53.59, -12.23, 75) mm, rotated rx 180 ry 0 rz -180 deg; joints [-164.2, -58.614, -83.559, 19.71, 53.835, -11.937]
  Call Extruder(16272.86585)
  MoveL 1666 to (54.97, 0, 75) mm, rotated rx -180 ry 0 rz 180 deg; joints [-162.641, -58.942, -82.66, 21.746, 53.642, -13.304]
  Call Extruder(16283.79607)
  MoveL 1667 to (53.59, 12.23, 75) mm, rotated rx -180 ry 0 rz 180 deg; joints [-160.996, -59.115, -82.189, 23.81, 53.764, -14.619]
  Call Extruder(16294.72622)
  MoveL 1668 to (49.52, 23.85, 75) mm, rotated rx -180 ry 0 rz -180 deg; joints [-159.322, -59.124, -82.166, 25.812, 54.19, -15.802]
  Call Extruder(16305.65649)
  MoveL 1669 to (42.98, 34.27, 75) mm, rotated rx -180 ry 0 rz -180 deg; joints [-157.673, -58.966, -82.594, 27.669, 54.894, -16.78]
  Call Extruder(16316.58662)
  MoveL 1670 to (34.27, 42.98, 75) mm, rotated rx 180 ry 0 rz 180 deg; joints [-156.102, -58.653, -83.452, 29.314, 55.836, -17.501]
  Call Extruder(16327.51689)
  MoveL 1671 to (23.85, 49.52, 75) mm, rotated rx 180 ry 0 rz 180 deg; joints [-154.667, -58.203, -84.701, 30.689, 56.965, -17.929]
  Call Extruder(16338.44704)
  MoveL 1672 to (12.23, 53.59, 75) mm, rotated rx 180 ry 0 rz 180 deg; joints [-153.426, -57.643, -86.285, 31.751, 58.224, -18.05]
  Call Extruder(16349.37726)
  MoveL 1673 to (0, 54.97, 75) mm, rotated rx 180 ry 0 rz 180 deg; joints [-152.438, -57.006, -88.133, 32.46, 59.555, -17.865]
  Call Extruder(16360.30748)
  MoveL 1674 to (-12.23, 53.59, 75) mm, rotated rx -180 ry 0 rz 180 deg; joints [-151.764, -56.328, -90.161, 32.784, 60.896, -17.394]
  Call Extruder(16371.23761)
  MoveL 1675 to (-23.85, 49.52, 75) mm, rotated rx 180 ry 0 rz 180 deg; joints [-151.463, -55.648, -92.273, 32.691, 62.188, -16.669]
  Call Extruder(16382.16789)
  MoveL 1676 to (-34.27, 42.98, 75) mm, rotated rx 180 ry 0 rz 180 deg; joints [-151.589, -55.001, -94.37, 32.155, 63.378, -15.733]
  Call Extruder(16393.09802)
  MoveL 1677 to (-42.98, 34.27, 75) mm, rotated rx -180 ry 0 rz -180 deg; joints [-152.179, -54.42, -96.347, 31.162, 64.411, -14.638]
  Call Extruder(16404.02829)
  MoveL 1678 to (-49.52, 23.85, 75) mm, rotated rx 180 ry 0 rz 180 deg; joints [-153.248, -53.931, -98.097, 29.717, 65.239, -13.445]
  Call Extruder(16414.95844)
  MoveL 1679 to (-53.59, 12.23, 75) mm, rotated rx 180 ry 0 rz -180 deg; joints [-154.769, -53.551, -99.522, 27.857, 65.817, -12.216]
  Call Extruder(16425.88866)
  MoveL 1680 to (-54.97, 0, 75) mm, rotated rx -180 ry 0 rz -180 deg; joints [-156.673, -53.292, -100.536, 25.664, 66.108, -11.013]
  Call Extruder(16431.41427)
  MoveL 1681 to (-54.27, -6.18, 75) mm, rotated rx -180 ry 0 rz 180 deg; joints [-157.76, -53.222, -100.817, 24.456, 66.097, -10.441]
  Set speed (130.0 mm/s)
  MoveL 1682 to (-49.9, -9.51, 75) mm, rotated rx 180 ry 0 rz 180 deg; joints [-158.616, -53.335, -100.364, 23.595, 65.633, -10.215]
  MoveL 1683 to (0.86, -13.23, 75) mm, rotated rx 180 ry 0 rz 180 deg; joints [-162.086, -55.537, -92.626, 20.832, 59.872, -10.813]
  Call Extruder(16434.73080)
  Set speed (80.0 mm/s)
  MoveL 1684 to (2.97, -12.99, 75) mm, rotated rx 180 ry 0 rz -180 deg; joints [-162.152, -55.649, -92.269, 20.808, 59.631, -10.876]
  Call Extruder(16439.39436)
  MoveL 1685 to (5.78, -12.01, 75) mm, rotated rx 180 ry 0 rz -180 deg; joints [-162.141, -55.813, -91.753, 20.895, 59.304, -11.028]
  Call Extruder(16444.05798)
  MoveL 1686 to (8.31, -10.42, 75) mm, rotated rx 180 ry 0 rz -180 deg; joints [-162.027, -55.973, -91.252, 21.098, 59.008, -11.237]
  Call Extruder(16448.72217)
  MoveL 1687 to (10.42, -8.31, 75) mm, rotated rx 180 ry 0 rz 180 deg; joints [-161.819, -56.123, -90.788, 21.404, 58.756, -11.492]
  Call Extruder(16453.38581)
  MoveL 1688 to (12.01, -5.78, 75) mm, rotated rx 180 ry 0 rz 180 deg; joints [-161.529, -56.254, -90.386, 21.798, 58.563, -11.783]
  Call Extruder(16458.04938)
  MoveL 1689 to (13, -2.97, 75) mm, rotated rx 180 ry 0 rz -180 deg; joints [-161.171, -56.36, -90.064, 22.259, 58.436, -12.092]
  Call Extruder(16462.71333)
  MoveL 1690 to (13.33, 0, 75) mm, rotated rx 180 ry 0 rz 180 deg; joints [-160.763, -56.434, -89.839, 22.762, 58.383, -12.405]
  Call Extruder(16467.37728)
  MoveL 1691 to (13, 2.97, 75) mm, rotated rx -180 ry 0 rz 180 deg; joints [-160.324, -56.473, -89.72, 23.284, 58.406, -12.705]
  Call Extruder(16472.04086)
  MoveL 1692 to (12.01, 5.78, 75) mm, rotated rx 180 ry 0 rz -180 deg; joints [-159.874, -56.475, -89.715, 23.8, 58.502, -12.977]
  Call Extruder(16476.70448)
  MoveL 1693 to (10.42, 8.31, 75) mm, rotated rx -180 ry 0 rz 180 deg; joints [-159.432, -56.44, -89.822, 24.286, 58.668, -13.205]
  Call Extruder(16481.36867)
  MoveL 1694 to (8.31, 10.42, 75) mm, rotated rx 180 ry 0 rz 180 deg; joints [-159.021, -56.369, -90.037, 24.718, 58.894, -13.378]
  Call Extruder(16486.03229)
  MoveL 1695 to (5.78, 12.01, 75) mm, rotated rx -180 ry 0 rz 180 deg; joints [-158.657, -56.266, -90.35, 25.078, 59.169, -13.487]
  Call Extruder(16490.69587)
  MoveL 1696 to (2.97, 12.99, 75) mm, rotated rx 180 ry 0 rz 180 deg; joints [-158.359, -56.137, -90.745, 25.347, 59.479, -13.527]
  Call Extruder(16495.35982)
  MoveL 1697 to (0, 13.33, 75) mm, rotated rx 180 ry 0 rz 180 deg; joints [-158.143, -55.989, -91.204, 25.513, 59.81, -13.496]
  Call Extruder(16500.02377)
  MoveL 1698 to (-2.97, 13, 75) mm, rotated rx 180 ry 0 rz 180 deg; joints [-158.019, -55.829, -91.703, 25.567, 60.145, -13.396]
  Call Extruder(16504.68734)
  MoveL 1699 to (-5.78, 12.01, 75) mm, rotated rx -180 ry 0 rz -180 deg; joints [-157.997, -55.665, -92.218, 25.506, 60.467, -13.234]
  Call Extruder(16509.35097)
  MoveL 1700 to (-8.31, 10.42, 75) mm, rotated rx -180 ry 0 rz -180 deg; joints [-158.08, -55.507, -92.723, 25.329, 60.761, -13.018]
  Call Extruder(16514.01517)
  MoveL 1701 to (-10.42, 8.31, 75) mm, rotated rx 180 ry 0 rz 180 deg; joints [-158.266, -55.361, -93.193, 25.045, 61.012, -12.759]
  Call Extruder(16518.67879)
  MoveL 1702 to (-12.01, 5.78, 75) mm, rotated rx -180 ry 0 rz -180 deg; joints [-158.549, -55.234, -93.603, 24.664, 61.209, -12.471]
  Call Extruder(16523.34236)
  MoveL 1703 to (-13, 2.97, 75) mm, rotated rx -180 ry 0 rz -180 deg; joints [-158.913, -55.133, -93.933, 24.206, 61.34, -12.167]
  Call Extruder(16528.00631)
  MoveL 1704 to (-13.33, 0, 75) mm, rotated rx 180 ry 0 rz 180 deg; joints [-159.341, -55.063, -94.166, 23.693, 61.398, -11.864]
  Call Extruder(16532.67027)
  MoveL 1705 to (-12.99, -2.97, 75) mm, rotated rx 180 ry 0 rz 180 deg; joints [-159.811, -55.026, -94.288, 23.151, 61.381, -11.575]
  Call Extruder(16537.33383)
  MoveL 1706 to (-12.01, -5.78, 75) mm, rotated rx 180 ry 0 rz -180 deg; joints [-160.294, -55.024, -94.294, 22.61, 61.289, -11.313]
  Call Extruder(16541.99746)
  MoveL 1707 to (-10.42, -8.31, 75) mm, rotated rx -180 ry 0 rz 180 deg; joints [-160.766, -55.058, -94.183, 22.098, 61.126, -11.093]
  Call Extruder(16546.66165)
  MoveL 1708 to (-8.31, -10.42, 75) mm, rotated rx 180 ry 0 rz -180 deg; joints [-161.2, -55.125, -93.961, 21.643, 60.9, -10.923]
  Call Extruder(16551.32529)
  MoveL 1709 to (-5.78, -12.01, 75) mm, rotated rx 180 ry 0 rz 180 deg; joints [-161.572, -55.223, -93.64, 21.271, 60.622, -10.812]
  Call Extruder(16555.98885)
  MoveL 1710 to (-2.97, -13, 75) mm, rotated rx 180 ry 0 rz 180 deg; joints [-161.863, -55.347, -93.236, 20.999, 60.307, -10.766]
  Call Extruder(16560.65279)
  MoveL 1711 to (0, -13.33, 75) mm, rotated rx 180 ry 0 rz -180 deg; joints [-162.059, -55.492, -92.771, 20.843, 59.971, -10.787]
  Call Extruder(16562.00024)
  MoveL 1712 to (0.86, -13.23, 75) mm, rotated rx 180 ry 0 rz 180 deg; joints [-162.086, -55.537, -92.626, 20.832, 59.872, -10.813]
  Set speed (130.0 mm/s)
  MoveL 1713 to (0.86, -13.23, 80) mm, rotated rx 180 ry 0 rz 180 deg; joints [-162.086, -54.77, -92.984, 20.917, 59.49, -10.981]
  MoveL 1714 to (-26.25, -4.54, 80) mm, rotated rx 180 ry 0 rz -180 deg; joints [-159.288, -53.591, -96.83, 23.498, 62.501, -11.351]
  Call Extruder(16564.23287)
  Set speed (60.0 mm/s)
  MoveL 1715 to (-26.09, -5.96, 80) mm, rotated rx 180 ry 0 rz 180 deg; joints [-159.522, -53.574, -96.888, 23.231, 62.494, -11.213]
  Call Extruder(16573.59765)
  MoveL 1716 to (-24.11, -11.61, 80) mm, rotated rx 180 ry 0 rz 180 deg; joints [-160.532, -53.57, -96.9, 22.111, 62.31, -10.691]
  Call Extruder(16582.96258)
  MoveL 1717 to (-20.93, -16.69, 80) mm, rotated rx 180 ry 0 rz 180 deg; joints [-161.513, -53.637, -96.672, 21.05, 61.982, -10.248]
  Call Extruder(16592.32778)
  MoveL 1718 to (-16.69, -20.93, 80) mm, rotated rx 180 ry 0 rz 180 deg; joints [-162.406, -53.771, -96.218, 20.112, 61.526, -9.903]
  Call Extruder(16601.69270)
  MoveL 1719 to (-11.61, -24.12, 80) mm, rotated rx -180 ry 0 rz 180 deg; joints [-163.159, -53.968, -95.563, 19.351, 60.966, -9.673]
  Call Extruder(16611.05749)
  MoveL 1720 to (-5.96, -26.09, 80) mm, rotated rx -180 ry 0 rz 180 deg; joints [-163.733, -54.218, -94.742, 18.807, 60.331, -9.569]
  Call Extruder(16620.42260)
  MoveL 1721 to (0, -26.77, 80) mm, rotated rx 180 ry 0 rz 180 deg; joints [-164.103, -54.511, -93.8, 18.505, 59.654, -9.598]
  Call Extruder(16623.02578)
  MoveL 1722 to (1.66, -26.58, 80) mm, rotated rx 180 ry 0 rz 180 deg; joints [-164.147, -54.6, -93.519, 18.491, 59.464, -9.643]
  Call Extruder(16629.78770)
  MoveL 1723 to (5.96, -26.09, 80) mm, rotated rx 180 ry 0 rz 180 deg; joints [-164.258, -54.834, -92.785, 18.458, 58.971, -9.762]
  Call Extruder(16639.15250)
  MoveL 1724 to (11.61, -24.11, 80) mm, rotated rx -180 ry 0 rz 180 deg; joints [-164.201, -55.169, -91.75, 18.66, 58.318, -10.058]
  Call Extruder(16648.51741)
  MoveL 1725 to (16.69, -20.93, 80) mm, rotated rx -180 ry 0 rz 180 deg; joints [-163.944, -55.501, -90.745, 19.094, 57.727, -10.472]
  Call Extruder(16657.88262)
  MoveL 1726 to (20.93, -16.69, 80) mm, rotated rx 180 ry 0 rz 180 deg; joints [-163.508, -55.811, -89.82, 19.732, 57.228, -10.988]
  Call Extruder(16667.24754)
  MoveL 1727 to (24.11, -11.61, 80) mm, rotated rx -180 ry 0 rz 180 deg; joints [-162.92, -56.084, -89.018, 20.538, 56.847, -11.578]
  Call Extruder(16676.61234)
  MoveL 1728 to (26.09, -5.96, 80) mm, rotated rx 180 ry 0 rz -180 deg; joints [-162.209, -56.304, -88.379, 21.468, 56.602, -12.214]
  Call Extruder(16685.97744)
  MoveL 1729 to (26.77, 0, 80) mm, rotated rx -180 ry 0 rz -180 deg; joints [-161.41, -56.46, -87.931, 22.475, 56.504, -12.861]
  Call Extruder(16695.34254)
  MoveL 1730 to (26.09, 5.96, 80) mm, rotated rx -180 ry 0 rz 180 deg; joints [-160.556, -56.542, -87.696, 23.511, 56.558, -13.482]
  Call Extruder(16704.70734)
  MoveL 1731 to (24.11, 11.61, 80) mm, rotated rx -180 ry 0 rz 180 deg; joints [-159.683, -56.546, -87.685, 24.528, 56.759, -14.044]
  Call Extruder(16714.07226)
  MoveL 1732 to (20.93, 16.69, 80) mm, rotated rx -180 ry 0 rz 180 deg; joints [-158.826, -56.471, -87.898, 25.482, 57.097, -14.515]
  Call Extruder(16723.43747)
  MoveL 1733 to (16.69, 20.93, 80) mm, rotated rx 180 ry 0 rz 180 deg; joints [-158.019, -56.323, -88.326, 26.33, 57.552, -14.87]
  Call Extruder(16732.80238)
  MoveL 1734 to (11.61, 24.11, 80) mm, rotated rx -180 ry 0 rz 180 deg; joints [-157.299, -56.108, -88.947, 27.037, 58.102, -15.092]
  Call Extruder(16742.16718)
  MoveL 1735 to (5.96, 26.09, 80) mm, rotated rx 180 ry 0 rz 180 deg; joints [-156.697, -55.84, -89.734, 27.573, 58.72, -15.17]
  Call Extruder(16751.53229)
  MoveL 1736 to (0, 26.77, 80) mm, rotated rx 180 ry 0 rz 180 deg; joints [-156.245, -55.533, -90.649, 27.912, 59.376, -15.102]
  Call Extruder(16760.89739)
  MoveL 1737 to (-5.96, 26.09, 80) mm, rotated rx 180 ry 0 rz 180 deg; joints [-155.969, -55.202, -91.648, 28.038, 60.037, -14.894]
  Call Extruder(16770.26218)
  MoveL 1738 to (-11.61, 24.11, 80) mm, rotated rx 180 ry 0 rz 180 deg; joints [-155.891, -54.867, -92.682, 27.938, 60.674, -14.56]
  Call Extruder(16779.62710)
  MoveL 1739 to (-16.69, 20.93, 80) mm, rotated rx 180 ry 0 rz -180 deg; joints [-156.025, -54.542, -93.701, 27.61, 61.256, -14.118]
  Call Extruder(16788.99231)
  MoveL 1740 to (-20.93, 16.69, 80) mm, rotated rx -180 ry 0 rz -180 deg; joints [-156.374, -54.246, -94.653, 27.061, 61.754, -13.592]
  Call Extruder(16798.35722)
  MoveL 1741 to (-24.11, 11.61, 80) mm, rotated rx 180 ry 0 rz 180 deg; joints [-156.928, -53.991, -95.488, 26.311, 62.145, -13.009]
  Call Extruder(16807.72202)
  MoveL 1742 to (-26.09, 5.96, 80) mm, rotated rx 180 ry 0 rz 180 deg; joints [-157.665, -53.788, -96.162, 25.391, 62.407, -12.399]
  Call Extruder(16817.08713)
  MoveL 1743 to (-26.77, 0, 80) mm, rotated rx 180 ry 0 rz 180 deg; joints [-158.546, -53.647, -96.637, 24.346, 62.526, -11.791]
  Call Extruder(16821.87586)
  MoveL 1744 to (-26.42, -3.05, 80) mm, rotated rx 180 ry 0 rz -180 deg; joints [-159.044, -53.609, -96.767, 23.777, 62.51, -11.495]
  Set speed (130.0 mm/s)
  MoveL 1745 to (-41.86, -6.29, 80) mm, rotated rx 180 ry 0 rz -180 deg; joints [-158.606, -52.882, -99.336, 23.885, 64.278, -10.879]
  Call Extruder(16826.87371)
  Set speed (60.0 mm/s)
  MoveL 1746 to (-41.5, -9.47, 80) mm, rotated rx 180 ry 0 rz 180 deg; joints [-159.151, -52.846, -99.468, 23.272, 64.265, -10.578]
  Call Extruder(16841.76935)
  MoveL 1747 to (-38.36, -18.47, 80) mm, rotated rx 180 ry 0 rz 180 deg; joints [-160.835, -52.841, -99.487, 21.426, 63.981, -9.768]
  Call Extruder(16856.66521)
  MoveL 1748 to (-33.29, -26.54, 80) mm, rotated rx -180 ry 0 rz 180 deg; joints [-162.466, -52.942, -99.116, 19.68, 63.461, -9.079]
  Call Extruder(16871.56103)
  MoveL 1749 to (-26.54, -33.28, 80) mm, rotated rx 180 ry 0 rz -180 deg; joints [-163.93, -53.147, -98.378, 18.145, 62.732, -8.539]
  Call Extruder(16886.45688)
  MoveL 1750 to (-18.47, -38.36, 80) mm, rotated rx -180 ry 0 rz 180 deg; joints [-165.137, -53.449, -97.316, 16.916, 61.833, -8.17]
  Call Extruder(16901.35253)
  MoveL 1751 to (-9.47, -41.5, 80) mm, rotated rx 180 ry 0 rz 180 deg; joints [-166.024, -53.839, -95.993, 16.059, 60.812, -7.991]
  Call Extruder(16916.24841)
  MoveL 1752 to (0, -42.57, 80) mm, rotated rx -180 ry 0 rz 180 deg; joints [-166.562, -54.299, -94.482, 15.61, 59.726, -8.017]
  Call Extruder(16921.61712)
  MoveL 1753 to (3.41, -42.19, 80) mm, rotated rx 180 ry 0 rz 180 deg; joints [-166.629, -54.48, -93.901, 15.596, 59.332, -8.103]
  Call Extruder(16931.14428)
  MoveL 1754 to (9.47, -41.5, 80) mm, rotated rx 180 ry 0 rz 180 deg; joints [-166.745, -54.809, -92.863, 15.577, 58.633, -8.256]
  Call Extruder(16946.03994)
  MoveL 1755 to (18.47, -38.36, 80) mm, rotated rx -180 ry 0 rz 180 deg; joints [-166.591, -55.343, -91.219, 15.943, 57.588, -8.706]
  Call Extruder(16960.93578)
  MoveL 1756 to (26.54, -33.29, 80) mm, rotated rx 180 ry 0 rz 180 deg; joints [-166.133, -55.876, -89.629, 16.675, 56.645, -9.352]
  Call Extruder(16975.83161)
  MoveL 1757 to (33.28, -26.54, 80) mm, rotated rx 180 ry 0 rz 180 deg; joints [-165.409, -56.377, -88.17, 17.721, 55.852, -10.169]
  Call Extruder(16990.72746)
  MoveL 1758 to (38.36, -18.47, 80) mm, rotated rx 180 ry 0 rz 180 deg; joints [-164.468, -56.818, -86.909, 19.021, 55.249, -11.117]
  Call Extruder(17005.62311)
  MoveL 1759 to (41.5, -9.47, 80) mm, rotated rx 180 ry 0 rz 180 deg; joints [-163.355, -57.176, -85.905, 20.504, 54.864, -12.146]
  Call Extruder(17020.51898)
  MoveL 1760 to (42.57, 0, 80) mm, rotated rx 180 ry 0 rz 180 deg; joints [-162.12, -57.429, -85.202, 22.094, 54.716, -13.196]
  Call Extruder(17035.41486)
  MoveL 1761 to (41.51, 9.47, 80) mm, rotated rx -180 ry 0 rz 180 deg; joints [-160.81, -57.563, -84.834, 23.716, 54.81, -14.207]
  Call Extruder(17050.31052)
  MoveL 1762 to (38.36, 18.47, 80) mm, rotated rx 180 ry 0 rz -180 deg; joints [-159.475, -57.569, -84.816, 25.297, 55.138, -15.118]
  Call Extruder(17065.20636)
  MoveL 1763 to (33.29, 26.54, 80) mm, rotated rx -180 ry 0 rz -180 deg; joints [-158.16, -57.448, -85.15, 26.771, 55.68, -15.878]
  Call Extruder(17080.10219)
  MoveL 1764 to (26.54, 33.28, 80) mm, rotated rx 180 ry 0 rz 180 deg; joints [-156.916, -57.206, -85.821, 28.079, 56.407, -16.445]
  Call Extruder(17094.99803)
  MoveL 1765 to (18.47, 38.36, 80) mm, rotated rx 180 ry 0 rz -180 deg; joints [-155.789, -56.858, -86.797, 29.172, 57.281, -16.791]
  Call Extruder(17109.89369)
  MoveL 1766 to (9.47, 41.51, 80) mm, rotated rx 180 ry 0 rz 180 deg; joints [-154.828, -56.423, -88.035, 30.009, 58.259, -16.901]
  Call Extruder(17124.78957)
  MoveL 1767 to (0, 42.57, 80) mm, rotated rx -180 ry 0 rz 180 deg; joints [-154.081, -55.927, -89.478, 30.556, 59.292, -16.777]
  Call Extruder(17139.68544)
  MoveL 1768 to (-9.47, 41.51, 80) mm, rotated rx 180 ry 0 rz 180 deg; joints [-153.594, -55.397, -91.057, 30.785, 60.334, -16.429]
  Call Extruder(17154.58109)
  MoveL 1769 to (-18.47, 38.36, 80) mm, rotated rx -180 ry 0 rz -180 deg; joints [-153.408, -54.861, -92.7, 30.674, 61.337, -15.881]
  Call Extruder(17169.47694)
  MoveL 1770 to (-26.54, 33.29, 80) mm, rotated rx -180 ry 0 rz 180 deg; joints [-153.557, -54.347, -94.325, 30.209, 62.255, -15.166]
  Call Extruder(17184.37276)
  MoveL 1771 to (-33.28, 26.54, 80) mm, rotated rx -180 ry 0 rz 180 deg; joints [-154.059, -53.881, -95.85, 29.39, 63.046, -14.322]
  Call Extruder(17199.26861)
  MoveL 1772 to (-38.36, 18.47, 80) mm, rotated rx -180 ry 0 rz -180 deg; joints [-154.913, -53.484, -97.195, 28.233, 63.673, -13.394]
  Call Extruder(17214.16427)
  MoveL 1773 to (-41.5, 9.47, 80) mm, rotated rx 180 ry 0 rz 180 deg; joints [-156.091, -53.173, -98.286, 26.778, 64.101, -12.431]
  Call Extruder(17229.06014)
  MoveL 1774 to (-42.57, 0, 80) mm, rotated rx 180 ry 0 rz -180 deg; joints [-157.533, -52.958, -99.059, 25.093, 64.304, -11.478]
  Call Extruder(17236.61442)
  MoveL 1775 to (-42.03, -4.8, 80) mm, rotated rx -180 ry 0 rz 180 deg; joints [-158.35, -52.899, -99.272, 24.172, 64.285, -11.021]
  Set speed (130.0 mm/s)
  MoveL 1776 to (-54.1, -7.67, 80) mm, rotated rx -180 ry 0 rz 180 deg; joints [-158.024, -52.374, -101.259, 24.247, 65.678, -10.509]
  Call Extruder(17240.68705)
  Set speed (30.0 mm/s)
  MoveL 1777 to (-53.59, -12.23, 80) mm, rotated rx 180 ry 0 rz -180 deg; joints [-158.835, -52.325, -101.451, 23.345, 65.664, -10.085]
  Call Extruder(17251.61718)
  MoveL 1778 to (-49.52, -23.85, 80) mm, rotated rx 180 ry 0 rz -180 deg; joints [-161.095, -52.318, -101.477, 20.892, 65.306, -9.06]
  Call Extruder(17262.54746)
  MoveL 1779 to (-42.98, -34.27, 80) mm, rotated rx 180 ry 0 rz 180 deg; joints [-163.275, -52.443, -100.988, 18.571, 64.637, -8.19]
  Call Extruder(17273.47758)
  MoveL 1780 to (-34.27, -42.98, 80) mm, rotated rx 180 ry 0 rz -180 deg; joints [-165.21, -52.698, -100.016, 16.545, 63.689, -7.501]
  Call Extruder(17284.40787)
  MoveL 1781 to (-23.85, -49.53, 80) mm, rotated rx 180 ry 0 rz 180 deg; joints [-166.774, -53.078, -98.624, 14.945, 62.517, -7.022]
  Call Extruder(17295.33800)
  MoveL 1782 to (-12.23, -53.59, 80) mm, rotated rx -180 ry 0 rz 180 deg; joints [-167.889, -53.571, -96.898, 13.854, 61.189, -6.778]
  Call Extruder(17306.26822)
  MoveL 1783 to (0, -54.97, 80) mm, rotated rx -180 ry 0 rz 180 deg; joints [-168.526, -54.159, -94.935, 13.309, 59.777, -6.791]
  Call Extruder(17314.47923)
  MoveL 1784 to (9.19, -53.93, 80) mm, rotated rx 180 ry 0 rz -180 deg; joints [-168.656, -54.648, -93.366, 13.308, 58.711, -7.004]
  Call Extruder(17317.19844)
  MoveL 1785 to (12.23, -53.59, 80) mm, rotated rx -180 ry 0 rz 180 deg; joints [-168.697, -54.815, -92.841, 13.31, 58.358, -7.075]
  Call Extruder(17328.12859)
  MoveL 1786 to (23.85, -49.53, 80) mm, rotated rx 180 ry 0 rz 180 deg; joints [-168.436, -55.508, -90.722, 13.828, 57.005, -7.634]
  Call Extruder(17339.05886)
  MoveL 1787 to (34.27, -42.98, 80) mm, rotated rx 180 ry 0 rz 180 deg; joints [-167.797, -56.2, -88.68, 14.81, 55.786, -8.456]
  Call Extruder(17349.98899)
  MoveL 1788 to (42.98, -34.27, 80) mm, rotated rx 180 ry 0 rz -180 deg; joints [-166.837, -56.854, -86.808, 16.189, 54.762, -9.509]
  Call Extruder(17360.91927)
  MoveL 1789 to (49.53, -23.85, 80) mm, rotated rx 180 ry 0 rz 180 deg; joints [-165.618, -57.432, -85.192, 17.883, 53.984, -10.743]
  Call Extruder(17371.84940)
  MoveL 1790 to (53.59, -12.23, 80) mm, rotated rx 180 ry 0 rz -180 deg; joints [-164.2, -57.901, -83.906, 19.801, 53.491, -12.09]
  Call Extruder(17382.77962)
  MoveL 1791 to (54.97, 0, 80) mm, rotated rx -180 ry 0 rz 180 deg; joints [-162.641, -58.234, -83.007, 21.845, 53.306, -13.471]
  Call Extruder(17393.70985)
  MoveL 1792 to (53.59, 12.23, 80) mm, rotated rx -180 ry 0 rz -180 deg; joints [-160.996, -58.409, -82.535, 23.918, 53.435, -14.8]
  Call Extruder(17404.63999)
  MoveL 1793 to (49.52, 23.85, 80) mm, rotated rx 180 ry 0 rz -180 deg; joints [-159.322, -58.418, -82.513, 25.926, 53.867, -15.995]
  Call Extruder(17415.57027)
  MoveL 1794 to (42.98, 34.27, 80) mm, rotated rx 180 ry 0 rz 180 deg; joints [-157.673, -58.258, -82.94, 27.788, 54.575, -16.986]
  Call Extruder(17426.50039)
  MoveL 1795 to (34.27, 42.98, 80) mm, rotated rx 180 ry 0 rz 180 deg; joints [-156.102, -57.941, -83.799, 29.436, 55.518, -17.718]
  Call Extruder(17437.43066)
  MoveL 1796 to (23.85, 49.52, 80) mm, rotated rx -180 ry 0 rz 180 deg; joints [-154.667, -57.484, -85.049, 30.813, 56.646, -18.156]
  Call Extruder(17448.36081)
  MoveL 1797 to (12.23, 53.59, 80) mm, rotated rx -180 ry 0 rz 180 deg; joints [-153.426, -56.916, -86.635, 31.875, 57.903, -18.284]
  Call Extruder(17459.29103)
  MoveL 1798 to (0, 54.97, 80) mm, rotated rx 180 ry 0 rz 180 deg; joints [-152.438, -56.268, -88.485, 32.583, 59.229, -18.107]
  Call Extruder(17470.22125)
  MoveL 1799 to (-12.23, 53.59, 80) mm, rotated rx 180 ry 0 rz 180 deg; joints [-151.764, -55.577, -90.515, 32.905, 60.562, -17.641]
  Call Extruder(17481.15139)
  MoveL 1800 to (-23.85, 49.52, 80) mm, rotated rx 180 ry 0 rz 180 deg; joints [-151.463, -54.883, -92.631, 32.808, 61.846, -16.919]
  Call Extruder(17492.08167)
  MoveL 1801 to (-34.27, 42.98, 80) mm, rotated rx -180 ry 0 rz 180 deg; joints [-151.589, -54.222, -94.732, 32.268, 63.024, -15.982]
  Call Extruder(17503.01179)
  MoveL 1802 to (-42.98, 34.27, 80) mm, rotated rx -180 ry 0 rz -180 deg; joints [-152.179, -53.626, -96.712, 31.269, 64.044, -14.885]
  Call Extruder(17513.94207)
  MoveL 1803 to (-49.52, 23.85, 80) mm, rotated rx 180 ry 0 rz 180 deg; joints [-153.248, -53.122, -98.466, 29.818, 64.858, -13.685]
  Call Extruder(17524.87221)
  MoveL 1804 to (-53.59, 12.23, 80) mm, rotated rx 180 ry 0 rz 180 deg; joints [-154.769, -52.731, -99.895, 27.952, 65.422, -12.446]
  Call Extruder(17535.80243)
  MoveL 1805 to (-54.97, 0, 80) mm, rotated rx 180 ry 0 rz -180 deg; joints [-156.673, -52.463, -100.912, 25.752, 65.7, -11.228]
  Call Extruder(17541.32805)
  MoveL 1806 to (-54.27, -6.18, 80) mm, rotated rx 180 ry 0 rz 180 deg; joints [-157.76, -52.39, -101.194, 24.54, 65.683, -10.648]
  Set speed (130.0 mm/s)
  MoveL 1807 to (-49.9, -9.51, 80) mm, rotated rx -180 ry 0 rz 180 deg; joints [-158.616, -52.508, -100.739, 23.678, 65.218, -10.415]
  MoveL 1808 to (0.16, -13.31, 80) mm, rotated rx -180 ry 0 rz 180 deg; joints [-162.064, -54.732, -93.102, 20.926, 59.569, -10.961]
  Call Extruder(17545.73953)
  Set speed (80.0 mm/s)
  MoveL 1809 to (2.97, -12.99, 80) mm, rotated rx 180 ry 0 rz -180 deg; joints [-162.152, -54.885, -92.626, 20.893, 59.25, -11.044]
  Call Extruder(17550.40310)
  MoveL 1810 to (5.78, -12.01, 80) mm, rotated rx 180 ry 0 rz 180 deg; joints [-162.141, -55.052, -92.11, 20.981, 58.926, -11.196]
  Call Extruder(17555.06672)
  MoveL 1811 to (8.31, -10.42, 80) mm, rotated rx -180 ry 0 rz -180 deg; joints [-162.027, -55.216, -91.607, 21.186, 58.633, -11.406]
  Call Extruder(17559.73092)
  MoveL 1812 to (10.42, -8.31, 80) mm, rotated rx 180 ry 0 rz 180 deg; joints [-161.819, -55.368, -91.143, 21.494, 58.384, -11.664]
  Call Extruder(17564.39455)
  MoveL 1813 to (12.01, -5.78, 80) mm, rotated rx 180 ry 0 rz -180 deg; joints [-161.529, -55.502, -90.74, 21.889, 58.194, -11.956]
  Call Extruder(17569.05811)
  MoveL 1814 to (12.99, -2.97, 80) mm, rotated rx 180 ry 0 rz -180 deg; joints [-161.171, -55.61, -90.418, 22.352, 58.07, -12.269]
  Call Extruder(17573.72207)
  MoveL 1815 to (13.33, 0, 80) mm, rotated rx 180 ry 0 rz 180 deg; joints [-160.763, -55.686, -90.192, 22.857, 58.019, -12.585]
  Call Extruder(17578.38602)
  MoveL 1816 to (13, 2.97, 80) mm, rotated rx 180 ry 0 rz 180 deg; joints [-160.324, -55.725, -90.074, 23.381, 58.044, -12.889]
  Call Extruder(17583.04959)
  MoveL 1817 to (12.01, 5.78, 80) mm, rotated rx 180 ry 0 rz -180 deg; joints [-159.874, -55.727, -90.068, 23.899, 58.142, -13.164]
  Call Extruder(17587.71322)
  MoveL 1818 to (10.42, 8.31, 80) mm, rotated rx -180 ry 0 rz 180 deg; joints [-159.432, -55.691, -90.176, 24.386, 58.308, -13.396]
  Call Extruder(17592.37741)
  MoveL 1819 to (8.31, 10.42, 80) mm, rotated rx 180 ry 0 rz -180 deg; joints [-159.021, -55.619, -90.391, 24.819, 58.534, -13.572]
  Call Extruder(17597.04103)
  MoveL 1820 to (5.78, 12.01, 80) mm, rotated rx 180 ry 0 rz 180 deg; joints [-158.657, -55.514, -90.705, 25.179, 58.809, -13.684]
  Call Extruder(17601.70461)
  MoveL 1821 to (2.97, 12.99, 80) mm, rotated rx 180 ry 0 rz 180 deg; joints [-158.359, -55.383, -91.1, 25.449, 59.118, -13.726]
  Call Extruder(17606.36856)
  MoveL 1822 to (0, 13.33, 80) mm, rotated rx -180 ry 0 rz 180 deg; joints [-158.143, -55.231, -91.559, 25.615, 59.448, -13.697]
  Call Extruder(17611.03251)
  MoveL 1823 to (-2.97, 13, 80) mm, rotated rx -180 ry 0 rz 180 deg; joints [-158.019, -55.068, -92.059, 25.669, 59.78, -13.598]
  Call Extruder(17615.69608)
  MoveL 1824 to (-5.78, 12.01, 80) mm, rotated rx -180 ry 0 rz 180 deg; joints [-157.997, -54.901, -92.575, 25.606, 60.1, -13.436]
  Call Extruder(17620.35971)
  MoveL 1825 to (-8.31, 10.42, 80) mm, rotated rx -180 ry 0 rz 180 deg; joints [-158.08, -54.739, -93.081, 25.428, 60.391, -13.219]
  Call Extruder(17625.02390)
  MoveL 1826 to (-10.42, 8.31, 80) mm, rotated rx -180 ry 0 rz 180 deg; joints [-158.266, -54.59, -93.552, 25.142, 60.639, -12.959]
  Call Extruder(17629.68753)
  MoveL 1827 to (-12.01, 5.78, 80) mm, rotated rx 180 ry 0 rz 180 deg; joints [-158.549, -54.46, -93.963, 24.76, 60.832, -12.669]
  Call Extruder(17634.35110)
  MoveL 1828 to (-12.99, 2.97, 80) mm, rotated rx 180 ry 0 rz -180 deg; joints [-158.913, -54.357, -94.294, 24.3, 60.96, -12.362]
  Call Extruder(17639.01505)
  MoveL 1829 to (-13.33, 0, 80) mm, rotated rx 180 ry 0 rz 180 deg; joints [-159.341, -54.285, -94.526, 23.785, 61.016, -12.055]
  Call Extruder(17643.67901)
  MoveL 1830 to (-12.99, -2.97, 80) mm, rotated rx 180 ry 0 rz 180 deg; joints [-159.811, -54.247, -94.649, 23.242, 60.997, -11.762]
  Call Extruder(17648.34257)
  MoveL 1831 to (-12.01, -5.78, 80) mm, rotated rx 180 ry 0 rz 180 deg; joints [-160.294, -54.245, -94.655, 22.699, 60.903, -11.497]
  Call Extruder(17653.00620)
  MoveL 1832 to (-10.42, -8.31, 80) mm, rotated rx 180 ry 0 rz -180 deg; joints [-160.766, -54.28, -94.544, 22.185, 60.739, -11.273]
  Call Extruder(17657.67039)
  MoveL 1833 to (-8.31, -10.42, 80) mm, rotated rx -180 ry 0 rz 180 deg; joints [-161.2, -54.348, -94.321, 21.73, 60.513, -11.099]
  Call Extruder(17662.33403)
  MoveL 1834 to (-5.78, -12.01, 80) mm, rotated rx 180 ry 0 rz 180 deg; joints [-161.572, -54.449, -94, 21.356, 60.236, -10.985]
  Call Extruder(17666.99759)
  MoveL 1835 to (-2.97, -12.99, 80) mm, rotated rx 180 ry 0 rz 180 deg; joints [-161.863, -54.576, -93.595, 21.084, 59.922, -10.936]
  Call Extruder(17671.66154)
  MoveL 1836 to (0, -13.33, 80) mm, rotated rx 180 ry 0 rz -180 deg; joints [-162.059, -54.723, -93.13, 20.928, 59.588, -10.956]
  Call Extruder(17671.91401)
  MoveL 1837 to (0.16, -13.31, 80) mm, rotated rx -180 ry 0 rz 180 deg; joints [-162.064, -54.732, -93.102, 20.926, 59.569, -10.961]
  Set speed (130.0 mm/s)
  MoveL 1838 to (0.16, -13.31, 85) mm, rotated rx -180 ry 0 rz 180 deg; joints [-162.064, -53.965, -93.451, 21.014, 59.179, -11.135]
  MoveL 1839 to (-26.25, -4.54, 85) mm, rotated rx 180 ry 0 rz 180 deg; joints [-159.288, -52.796, -97.186, 23.59, 62.099, -11.549]
  Call Extruder(17674.14663)
  Set speed (60.0 mm/s)
  MoveL 1840 to (-26.09, -5.96, 85) mm, rotated rx -180 ry 0 rz -180 deg; joints [-159.522, -52.778, -97.244, 23.322, 62.09, -11.409]
  Call Extruder(17683.51142)
  MoveL 1841 to (-24.11, -11.61, 85) mm, rotated rx -180 ry 0 rz 180 deg; joints [-160.532, -52.775, -97.256, 22.198, 61.903, -10.879]
  Call Extruder(17692.87634)
  MoveL 1842 to (-20.93, -16.69, 85) mm, rotated rx 180 ry 0 rz -180 deg; joints [-161.513, -52.843, -97.028, 21.135, 61.573, -10.427]
  Call Extruder(17702.24155)
  MoveL 1843 to (-16.69, -20.93, 85) mm, rotated rx 180 ry 0 rz 180 deg; joints [-162.406, -52.981, -96.573, 20.194, 61.117, -10.074]
  Call Extruder(17711.60647)
  MoveL 1844 to (-11.61, -24.12, 85) mm, rotated rx 180 ry 0 rz 180 deg; joints [-163.159, -53.183, -95.916, 19.431, 60.559, -9.837]
  Call Extruder(17720.97126)
  MoveL 1845 to (-5.96, -26.09, 85) mm, rotated rx -180 ry 0 rz 180 deg; joints [-163.733, -53.439, -95.094, 18.886, 59.927, -9.728]
  Call Extruder(17730.33637)
  MoveL 1846 to (0, -26.77, 85) mm, rotated rx 180 ry 0 rz 180 deg; joints [-164.103, -53.739, -94.15, 18.585, 59.254, -9.754]
  Call Extruder(17735.34658)
  MoveL 1847 to (3.19, -26.41, 85) mm, rotated rx 180 ry 0 rz 180 deg; joints [-164.187, -53.914, -93.607, 18.559, 58.892, -9.841]
  Call Extruder(17739.70146)
  MoveL 1848 to (5.96, -26.09, 85) mm, rotated rx 180 ry 0 rz 180 deg; joints [-164.258, -54.069, -93.133, 18.538, 58.576, -9.917]
  Call Extruder(17749.06627)
  MoveL 1849 to (11.61, -24.11, 85) mm, rotated rx 180 ry 0 rz 180 deg; joints [-164.201, -54.411, -92.096, 18.742, 57.928, -10.213]
  Call Extruder(17758.43118)
  MoveL 1850 to (16.69, -20.93, 85) mm, rotated rx -180 ry 0 rz 180 deg; joints [-163.944, -54.749, -91.09, 19.179, 57.343, -10.63]
  Call Extruder(17767.79639)
  MoveL 1851 to (20.93, -16.69, 85) mm, rotated rx 180 ry 0 rz 180 deg; joints [-163.508, -55.066, -90.164, 19.82, 56.85, -11.149]
  Call Extruder(17777.16131)
  MoveL 1852 to (24.12, -11.61, 85) mm, rotated rx -180 ry 0 rz 180 deg; joints [-162.92, -55.344, -89.361, 20.63, 56.475, -11.746]
  Call Extruder(17786.52610)
  MoveL 1853 to (26.09, -5.96, 85) mm, rotated rx -180 ry 0 rz -180 deg; joints [-162.209, -55.568, -88.721, 21.564, 56.235, -12.388]
  Call Extruder(17795.89121)
  MoveL 1854 to (26.77, 0, 85) mm, rotated rx 180 ry 0 rz -180 deg; joints [-161.41, -55.726, -88.273, 22.575, 56.142, -13.041]
  Call Extruder(17805.25631)
  MoveL 1855 to (26.09, 5.96, 85) mm, rotated rx -180 ry 0 rz 180 deg; joints [-160.556, -55.809, -88.038, 23.615, 56.2, -13.67]
  Call Extruder(17814.62111)
  MoveL 1856 to (24.12, 11.61, 85) mm, rotated rx -180 ry 0 rz -180 deg; joints [-159.683, -55.813, -88.027, 24.635, 56.404, -14.238]
  Call Extruder(17823.98602)
  MoveL 1857 to (20.93, 16.69, 85) mm, rotated rx -180 ry 0 rz -180 deg; joints [-158.826, -55.738, -88.24, 25.592, 56.743, -14.716]
  Call Extruder(17833.35123)
  MoveL 1858 to (16.69, 20.93, 85) mm, rotated rx 180 ry 0 rz 180 deg; joints [-158.019, -55.587, -88.668, 26.442, 57.199, -15.078]
  Call Extruder(17842.71615)
  MoveL 1859 to (11.61, 24.11, 85) mm, rotated rx -180 ry 0 rz 180 deg; joints [-157.299, -55.369, -89.29, 27.15, 57.749, -15.305]
  Call Extruder(17852.08095)
  MoveL 1860 to (5.96, 26.09, 85) mm, rotated rx 180 ry 0 rz 180 deg; joints [-156.697, -55.096, -90.078, 27.686, 58.365, -15.388]
  Call Extruder(17861.44605)
  MoveL 1861 to (0, 26.77, 85) mm, rotated rx 180 ry 0 rz 180 deg; joints [-156.245, -54.782, -90.994, 28.026, 59.017, -15.324]
  Call Extruder(17870.81115)
  MoveL 1862 to (-5.96, 26.09, 85) mm, rotated rx 180 ry 0 rz 180 deg; joints [-155.969, -54.445, -91.994, 28.15, 59.675, -15.118]
  Call Extruder(17880.17595)
  MoveL 1863 to (-11.61, 24.11, 85) mm, rotated rx 180 ry 0 rz 180 deg; joints [-155.891, -54.102, -93.031, 28.048, 60.307, -14.784]
  Call Extruder(17889.54087)
